KUKA KRL program: EPS_2_251529_SANMH_A_20250926032654.src

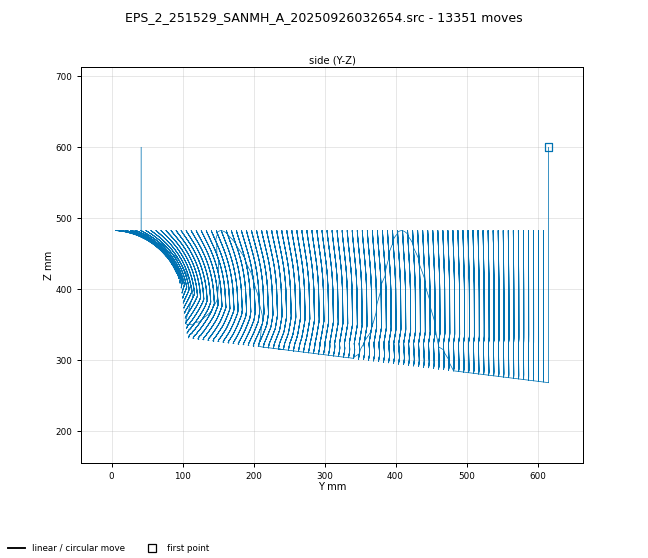
[picture p0: tool path of EPS_2_251529_SANMH_A_20250926032654.src, 13351 of 13353 moves have a stored position in this frame; points joined in program order, loops and branches not executed]
&ACCESS RVP
&REL 4
&COMMENT QRS 19112012
&PARAM EDITMASK = *
DEF PART()
EXT BAS (BAS_COMMAND :IN,REAL :IN )
INT I
BAS (#INITMOV,0 )

;KUKA QRS Post kuka4.cps  Date:22-06-2017 !

File_ID=2851

QRS_PRE_INIT()

;Init var - Until changes are made in qrs_pre_init
Outlet_Square_prg=0
Inlet_1_Square_prg=0
Inlet_2_Square_prg=0
Inlet_3_Square_prg=0
Inlet_4_Square_prg=0
Inlet_5_Square_prg=0

Outlet_1={X 0.000, Y 541.230, Z 408.000, B 0.000, E1 0.000 }
Inlet_1={X 0.000, Y 541.230, Z 408.000, B 0.000, E1 180.000 }
Outlet_1_type=150
Inlet_1_type=150
;QRS#1=Sidecore dimensions
;QRS#2=150-6" PVC SDR 28
;QRS#3=150-6" PVC SDR 28
;QRS#4=
;QRS#5=
;QRS#6=
;QRS#7=
;QRS#8=
;QRS#9=10-06 PSX
;QRS#10=10-06 PSX
;QRS#11=
;QRS#12=
;QRS#13=
;QRS#14=
;QRS#15=
;QRS#16=1220x127x762 2,5'
;QRS#17=EPS Height
;QRS#18=483
;QRS#19=*
;QRS#20= UPDATED VERSION 22-06-2017
;QRS#21=*
Outlet_Square=070
Inlet_1_Square=070
Inlet_2_Square=0
Inlet_3_Square=0
Inlet_4_Square=0
Inlet_5_Square=0
Mill_Square=1
Outlet_Square_Prg=203
Inlet_1_Square_prg=203

QRS_INIT()

$ADVANCE=5

; T1
PTP {E1 173.65,E2 173.65}
PTP {X 0,Y 615.436,A -85,B 0,C 180,E1 173.65,E2 173.65,E3 0,E4 0,E5 0,E6 0}
QRS_SPEED_INIT()
LIN {X 0,Y 615.436,Z 600,A -85,B 0,C 180,E1 173.65,E2 173.65,E3 0,E4 0,E5 0,E6 0} C_VEL
LIN {X 0,Y 615.436,Z 278.69,A -85,B 0,C 180,E1 173.65,E2 173.65} C_VEL
LIN {X 0,Y 615.436,Z 270.512,A -85,B 0,C 180,E1 173.65,E2 173.65} C_VEL
LIN {X 0,Y 615.421,Z 268.512,A -85,B 0,C 180,E1 173.464,E2 173.464} C_VEL
LIN {X 0,Y 615.418,Z 268.512,A -85,B 0,C 180,E1 171.462,E2 171.462} C_VEL
LIN {X 0,Y 615.412,Z 268.512,A -85,B 0,C 180,E1 169.141,E2 169.141} C_VEL
LIN {X 0,Y 615.434,Z 268.512,A -85,B 0,C 180,E1 166.798,E2 166.798} C_VEL
LIN {X 0,Y 615.46,Z 268.512,A -85,B 0,C 180,E1 164.094,E2 164.094} C_VEL
LIN {X 0,Y 615.413,Z 268.512,A -85,B 0,C 180,E1 161.352,E2 161.352} C_VEL
LIN {X 0,Y 615.489,Z 268.512,A -85,B 0,C 180,E1 158.568,E2 158.568} C_VEL
LIN {X 0,Y 615.416,Z 268.512,A -85,B 0,C 180,E1 155.725,E2 155.725} C_VEL
LIN {X 0,Y 615.415,Z 268.512,A -85,B 0,C 180,E1 153.552,E2 153.552} C_VEL
LIN {X 0,Y 615.478,Z 268.514,A -85,B 0,C 180,E1 150.593,E2 150.593} C_VEL
LIN {X 0,Y 615.446,Z 268.511,A -85,B 0,C 180,E1 148.312,E2 148.312} C_VEL
LIN {X 0,Y 615.418,Z 268.511,A -85,B 0,C 180,E1 145.974,E2 145.974} C_VEL
LIN {X 0,Y 615.472,Z 268.512,A -85,B 0,C 180,E1 143.064,E2 143.064} C_VEL
LIN {X 0,Y 615.424,Z 268.511,A -85,B 0,C 180,E1 140.245,E2 140.245} C_VEL
LIN {X 0,Y 615.417,Z 268.511,A -85,B 0,C 180,E1 137.926,E2 137.926} C_VEL
LIN {X 0,Y 615.42,Z 268.512,A -85,B 0,C 180,E1 135.844,E2 135.844} C_VEL
LIN {X 0,Y 615.48,Z 268.512,A -85,B 0,C 180,E1 133.244,E2 133.244} C_VEL
LIN {X 0,Y 615.438,Z 268.51,A -85,B 0,C 180,E1 130.609,E2 130.609} C_VEL
LIN {X 0,Y 615.466,Z 268.51,A -85,B 0,C 180,E1 128.905,E2 128.905} C_VEL
LIN {X 0,Y 615.423,Z 268.51,A -85,B 0,C 180,E1 126.428,E2 126.428} C_VEL
LIN {X 0,Y 615.471,Z 268.513,A -85,B 0,C 180,E1 123.532,E2 123.532} C_VEL
LIN {X 0,Y 615.448,Z 268.509,A -85,B 0,C 180,E1 120.921,E2 120.921} C_VEL
LIN {X 0,Y 615.421,Z 268.51,A -85,B 0,C 180,E1 118.439,E2 118.439} C_VEL
LIN {X 0,Y 615.474,Z 268.512,A -85,B 0,C 180,E1 115.716,E2 115.716} C_VEL
LIN {X 0,Y 615.43,Z 268.509,A -85,B 0,C 180,E1 112.846,E2 112.846} C_VEL
LIN {X 0,Y 615.423,Z 268.51,A -85,B 0,C 180,E1 110.54,E2 110.54} C_VEL
LIN {X 0,Y 615.492,Z 268.765,A -85,B 0,C 180,E1 109.598,E2 109.598} C_VEL
LIN {X 0,Y 615.471,Z 283.781,A -85,B 0,C 180,E1 106.928,E2 106.928} C_VEL
LIN {X 0,Y 615.47,Z 299.164,A -85,B 0,C 180,E1 104.241,E2 104.241} C_VEL
LIN {X 0,Y 615.494,Z 314.868,A -85,B 0,C 180,E1 101.526,E2 101.526} C_VEL
LIN {X 0,Y 615.495,Z 323.333,A -85,B 0,C 180,E1 100.111,E2 100.111} C_VEL
LIN {X 0,Y 615.495,Z 324.837,A -85,B 0,C 180,E1 100.049,E2 100.049} C_VEL
LIN {X 0,Y 615.492,Z 399.723,A -85,B 0,C 180,E1 99.157,E2 99.157} C_VEL
LIN {X 0,Y 615.496,Z 407.902,A -85,B 0,C 180,E1 98.991,E2 98.991} C_VEL
LIN {X 0,Y 615.497,Z 416.457,A -85,B 0,C 180,E1 98.743,E2 98.743} C_VEL
LIN {X 0,Y 615.497,Z 424.066,A -85,B 0,C 180,E1 98.454,E2 98.454} C_VEL
LIN {X 0,Y 615.499,Z 432.585,A -85,B 0,C 180,E1 98.04,E2 98.04} C_VEL
LIN {X 0,Y 615.487,Z 440.752,A -85,B 0,C 180,E1 97.545,E2 97.545} C_VEL
LIN {X 0,Y 615.492,Z 447.39,A -85,B 0,C 180,E1 97.058,E2 97.058} C_VEL
LIN {X 0,Y 615.498,Z 453.186,A -85,B 0,C 180,E1 96.556,E2 96.556} C_VEL
LIN {X 0,Y 615.499,Z 459.536,A -85,B 0,C 180,E1 95.898,E2 95.898} C_VEL
LIN {X 0,Y 615.495,Z 465.985,A -85,B 0,C 180,E1 95.077,E2 95.077} C_VEL
LIN {X 0,Y 615.491,Z 471.123,A -85,B 0,C 180,E1 94.256,E2 94.256} C_VEL
LIN {X 0,Y 615.493,Z 475.887,A -85,B 0,C 180,E1 93.273,E2 93.273} C_VEL
LIN {X 0,Y 615.493,Z 478.2,A -85,B 0,C 180,E1 92.618,E2 92.618} C_VEL
LIN {X 0,Y 615.5,Z 479.976,A -85,B 0,C 180,E1 91.963,E2 91.963} C_VEL
LIN {X 0,Y 615.492,Z 481.266,A -85,B 0,C 180,E1 91.309,E2 91.309} C_VEL
LIN {X 0,Y 615.491,Z 482.084,A -85,B 0,C 180,E1 90.654,E2 90.654} C_VEL
LIN {X 0,Y 615.492,Z 482.384,A -85,B 0,C 180,E1 90,E2 90} C_VEL
LIN {X 0,Y 615.492,Z 482.125,A -85,B 0,C 180,E1 89.346,E2 89.346} C_VEL
LIN {X 0,Y 615.494,Z 481.394,A -85,B 0,C 180,E1 88.691,E2 88.691} C_VEL
LIN {X 0,Y 615.5,Z 480.194,A -85,B 0,C 180,E1 88.037,E2 88.037} C_VEL
LIN {X 0,Y 615.49,Z 477.376,A -85,B 0,C 180,E1 87.055,E2 87.055} C_VEL
LIN {X 0,Y 615.492,Z 474.81,A -85,B 0,C 180,E1 86.399,E2 86.399} C_VEL
LIN {X 0,Y 615.495,Z 469.743,A -85,B 0,C 180,E1 85.416,E2 85.416} C_VEL
LIN {X 0,Y 615.496,Z 464.288,A -85,B 0,C 180,E1 84.595,E2 84.595} C_VEL
LIN {X 0,Y 615.497,Z 457.454,A -85,B 0,C 180,E1 83.773,E2 83.773} C_VEL
LIN {X 0,Y 615.497,Z 450.42,A -85,B 0,C 180,E1 83.1,E2 83.1} C_VEL
LIN {X 0,Y 615.487,Z 442.074,A -85,B 0,C 180,E1 82.455,E2 82.455} C_VEL
LIN {X 0,Y 615.499,Z 434.197,A -85,B 0,C 180,E1 81.96,E2 81.96} C_VEL
LIN {X 0,Y 615.497,Z 426.076,A -85,B 0,C 180,E1 81.546,E2 81.546} C_VEL
LIN {X 0,Y 615.497,Z 417.865,A -85,B 0,C 180,E1 81.216,E2 81.216} C_VEL
LIN {X 0,Y 615.497,Z 409.844,A -85,B 0,C 180,E1 80.967,E2 80.967} C_VEL
LIN {X 0,Y 615.497,Z 400.169,A -85,B 0,C 180,E1 80.76,E2 80.76} C_VEL
LIN {X 0,Y 615.493,Z 324.19,A -85,B 0,C 180,E1 79.848,E2 79.848} C_VEL
LIN {X 0,Y 615.49,Z 322.717,A -85,B 0,C 180,E1 79.723,E2 79.723} C_VEL
LIN {X 0,Y 615.485,Z 307.623,A -85,B 0,C 180,E1 77.135,E2 77.135} C_VEL
LIN {X 0,Y 615.491,Z 292.071,A -85,B 0,C 180,E1 74.435,E2 74.435} C_VEL
LIN {X 0,Y 615.479,Z 276.618,A -85,B 0,C 180,E1 71.719,E2 71.719} C_VEL
LIN {X 0,Y 615.493,Z 268.624,A -85,B 0,C 180,E1 70.272,E2 70.272} C_VEL
LIN {X 0,Y 615.436,Z 268.51,A -85,B 0,C 180,E1 67.666,E2 67.666} C_VEL
LIN {X 0,Y 615.437,Z 268.51,A -85,B 0,C 180,E1 65.726,E2 65.726} C_VEL
LIN {X 0,Y 615.427,Z 268.509,A -85,B 0,C 180,E1 63.554,E2 63.554} C_VEL
LIN {X 0,Y 615.431,Z 268.508,A -85,B 0,C 180,E1 61.34,E2 61.34} C_VEL
LIN {X 0,Y 615.469,Z 268.507,A -85,B 0,C 180,E1 58.917,E2 58.917} C_VEL
LIN {X 0,Y 615.435,Z 268.51,A -85,B 0,C 180,E1 55.976,E2 55.976} C_VEL
LIN {X 0,Y 615.428,Z 268.509,A -85,B 0,C 180,E1 53.572,E2 53.572} C_VEL
LIN {X 0,Y 615.49,Z 268.507,A -85,B 0,C 180,E1 50.938,E2 50.938} C_VEL
LIN {X 0,Y 615.467,Z 268.512,A -85,B 0,C 180,E1 48.526,E2 48.526} C_VEL
LIN {X 0,Y 615.425,Z 268.51,A -85,B 0,C 180,E1 46.009,E2 46.009} C_VEL
LIN {X 0,Y 615.424,Z 268.51,A -85,B 0,C 180,E1 43.993,E2 43.993} C_VEL
LIN {X 0,Y 615.449,Z 268.508,A -85,B 0,C 180,E1 41.477,E2 41.477} C_VEL
LIN {X 0,Y 615.485,Z 268.512,A -85,B 0,C 180,E1 38.905,E2 38.905} C_VEL
LIN {X 0,Y 615.43,Z 268.511,A -85,B 0,C 180,E1 36.429,E2 36.429} C_VEL
LIN {X 0,Y 615.422,Z 268.51,A -85,B 0,C 180,E1 34.026,E2 34.026} C_VEL
LIN {X 0,Y 615.445,Z 268.51,A -85,B 0,C 180,E1 31.688,E2 31.688} C_VEL
LIN {X 0,Y 615.479,Z 268.511,A -85,B 0,C 180,E1 29.407,E2 29.407} C_VEL
LIN {X 0,Y 615.42,Z 268.511,A -85,B 0,C 180,E1 26.447,E2 26.447} C_VEL
LIN {X 0,Y 615.435,Z 268.51,A -85,B 0,C 180,E1 24,E2 24} C_VEL
LIN {X 0,Y 615.498,Z 268.513,A -85,B 0,C 180,E1 21.432,E2 21.432} C_VEL
LIN {X 0,Y 615.415,Z 268.512,A -85,B 0,C 180,E1 18.589,E2 18.589} C_VEL
LIN {X 0,Y 615.462,Z 268.51,A -85,B 0,C 180,E1 15.906,E2 15.906} C_VEL
LIN {X 0,Y 615.441,Z 268.512,A -85,B 0,C 180,E1 13.202,E2 13.202} C_VEL
LIN {X 0,Y 615.417,Z 268.512,A -85,B 0,C 180,E1 10.861,E2 10.861} C_VEL
LIN {X 0,Y 615.421,Z 268.511,A -85,B 0,C 180,E1 8.538,E2 8.538} C_VEL
LIN {X 0,Y 615.496,Z 268.511,A -85,B 0,C 180,E1 5.899,E2 5.899} C_VEL
LIN {X 0,Y 615.426,Z 268.512,A -85,B 0,C 180,E1 3.273,E2 3.273} C_VEL
LIN {X 0,Y 615.425,Z 268.512,A -85,B 0,C 180,E1 1.309,E2 1.309} C_VEL
LIN {X 0,Y 615.423,Z 268.512,A -85,B 0,C 180,E1 -0.654,E2 -0.654} C_VEL
LIN {X 0,Y 615.42,Z 268.513,A -85,B 0,C 180,E1 -2.618,E2 -2.618} C_VEL
LIN {X 0,Y 615.42,Z 268.513,A -85,B 0,C 180,E1 -4.585,E2 -4.585} C_VEL
LIN {X 0,Y 615.42,Z 268.512,A -85,B 0,C 180,E1 -6.557,E2 -6.557} C_VEL
LIN {X 0,Y 615.418,Z 268.512,A -85,B 0,C 180,E1 -8.538,E2 -8.538} C_VEL
LIN {X 0,Y 615.413,Z 268.512,A -85,B 0,C 180,E1 -10.859,E2 -10.859} C_VEL
LIN {X 0,Y 615.435,Z 268.512,A -85,B 0,C 180,E1 -13.202,E2 -13.202} C_VEL
LIN {X 0,Y 615.46,Z 268.512,A -85,B 0,C 180,E1 -15.906,E2 -15.906} C_VEL
LIN {X 0,Y 615.414,Z 268.512,A -85,B 0,C 180,E1 -18.648,E2 -18.648} C_VEL
LIN {X 0,Y 615.491,Z 268.512,A -85,B 0,C 180,E1 -21.432,E2 -21.432} C_VEL
LIN {X 0,Y 615.418,Z 268.512,A -85,B 0,C 180,E1 -24.275,E2 -24.275} C_VEL
LIN {X 0,Y 615.416,Z 268.512,A -85,B 0,C 180,E1 -26.447,E2 -26.447} C_VEL
LIN {X 0,Y 615.479,Z 268.513,A -85,B 0,C 180,E1 -29.407,E2 -29.407} C_VEL
LIN {X 0,Y 615.447,Z 268.51,A -85,B 0,C 180,E1 -31.688,E2 -31.688} C_VEL
LIN {X 0,Y 615.421,Z 268.511,A -85,B 0,C 180,E1 -34.026,E2 -34.026} C_VEL
LIN {X 0,Y 615.475,Z 268.512,A -85,B 0,C 180,E1 -36.937,E2 -36.937} C_VEL
LIN {X 0,Y 615.426,Z 268.511,A -85,B 0,C 180,E1 -39.755,E2 -39.755} C_VEL
LIN {X 0,Y 615.42,Z 268.511,A -85,B 0,C 180,E1 -42.075,E2 -42.075} C_VEL
LIN {X 0,Y 615.423,Z 268.511,A -85,B 0,C 180,E1 -44.155,E2 -44.155} C_VEL
LIN {X 0,Y 615.485,Z 268.512,A -85,B 0,C 180,E1 -46.756,E2 -46.756} C_VEL
LIN {X 0,Y 615.44,Z 268.509,A -85,B 0,C 180,E1 -49.391,E2 -49.391} C_VEL
LIN {X 0,Y 615.467,Z 268.509,A -85,B 0,C 180,E1 -51.095,E2 -51.095} C_VEL
LIN {X 0,Y 615.425,Z 268.51,A -85,B 0,C 180,E1 -53.572,E2 -53.572} C_VEL
LIN {X 0,Y 615.479,Z 268.512,A -85,B 0,C 180,E1 -56.467,E2 -56.467} C_VEL
LIN {X 0,Y 615.449,Z 268.508,A -85,B 0,C 180,E1 -59.079,E2 -59.079} C_VEL
LIN {X 0,Y 615.424,Z 268.51,A -85,B 0,C 180,E1 -61.561,E2 -61.561} C_VEL
LIN {X 0,Y 615.498,Z 268.512,A -85,B 0,C 180,E1 -64.429,E2 -64.429} C_VEL
LIN {X 0,Y 615.432,Z 268.509,A -85,B 0,C 180,E1 -67.154,E2 -67.154} C_VEL
LIN {X 0,Y 615.427,Z 268.51,A -85,B 0,C 180,E1 -69.458,E2 -69.458} C_VEL
LIN {X 0,Y 615.492,Z 268.773,A -85,B 0,C 180,E1 -70.359,E2 -70.359} C_VEL
LIN {X 0,Y 615.469,Z 284.037,A -85,B 0,C 180,E1 -73.072,E2 -73.072} C_VEL
LIN {X 0,Y 615.471,Z 299.417,A -85,B 0,C 180,E1 -75.758,E2 -75.758} C_VEL
LIN {X 0,Y 615.492,Z 315.131,A -85,B 0,C 180,E1 -78.474,E2 -78.474} C_VEL
LIN {X 0,Y 615.494,Z 323.371,A -85,B 0,C 180,E1 -79.848,E2 -79.848} C_VEL
LIN {X 0,Y 615.494,Z 325.037,A -85,B 0,C 180,E1 -79.91,E2 -79.91} C_VEL
LIN {X 0,Y 615.494,Z 399.946,A -85,B 0,C 180,E1 -80.802,E2 -80.802} C_VEL
LIN {X 0,Y 615.497,Z 409.7,A -85,B 0,C 180,E1 -81.009,E2 -81.009} C_VEL
LIN {X 0,Y 615.499,Z 420.157,A -85,B 0,C 180,E1 -81.34,E2 -81.34} C_VEL
LIN {X 0,Y 615.497,Z 430.43,A -85,B 0,C 180,E1 -81.794,E2 -81.794} C_VEL
LIN {X 0,Y 615.489,Z 440.201,A -85,B 0,C 180,E1 -82.372,E2 -82.372} C_VEL
LIN {X 0,Y 615.494,Z 447.936,A -85,B 0,C 180,E1 -82.942,E2 -82.942} C_VEL
LIN {X 0,Y 615.497,Z 455.335,A -85,B 0,C 180,E1 -83.608,E2 -83.608} C_VEL
LIN {X 0,Y 615.498,Z 462.738,A -85,B 0,C 180,E1 -84.43,E2 -84.43} C_VEL
LIN {X 0,Y 615.497,Z 468.533,A -85,B 0,C 180,E1 -85.252,E2 -85.252} C_VEL
LIN {X 0,Y 615.496,Z 473.1,A -85,B 0,C 180,E1 -86.072,E2 -86.072} C_VEL
LIN {X 0,Y 615.492,Z 476.069,A -85,B 0,C 180,E1 -86.727,E2 -86.727} C_VEL
LIN {X 0,Y 615.494,Z 478.357,A -85,B 0,C 180,E1 -87.382,E2 -87.382} C_VEL
LIN {X 0,Y 615.5,Z 480.085,A -85,B 0,C 180,E1 -88.037,E2 -88.037} C_VEL
LIN {X 0,Y 615.493,Z 481.33,A -85,B 0,C 180,E1 -88.691,E2 -88.691} C_VEL
LIN {X 0,Y 615.491,Z 482.104,A -85,B 0,C 180,E1 -89.346,E2 -89.346} C_VEL
LIN {X 0,Y 615.491,Z 482.389,A -85,B 0,C 180,E1 -90,E2 -90} C_VEL
LIN {X 0,Y 615.491,Z 482.104,A -85,B 0,C 180,E1 -90.654,E2 -90.654} C_VEL
LIN {X 0,Y 615.493,Z 481.33,A -85,B 0,C 180,E1 -91.309,E2 -91.309} C_VEL
LIN {X 0,Y 615.5,Z 480.085,A -85,B 0,C 180,E1 -91.963,E2 -91.963} C_VEL
LIN {X 0,Y 615.488,Z 477.221,A -85,B 0,C 180,E1 -92.945,E2 -92.945} C_VEL
LIN {X 0,Y 615.491,Z 474.604,A -85,B 0,C 180,E1 -93.601,E2 -93.601} C_VEL
LIN {X 0,Y 615.495,Z 469.483,A -85,B 0,C 180,E1 -94.584,E2 -94.584} C_VEL
LIN {X 0,Y 615.495,Z 463.969,A -85,B 0,C 180,E1 -95.405,E2 -95.405} C_VEL
LIN {X 0,Y 615.498,Z 457.019,A -85,B 0,C 180,E1 -96.227,E2 -96.227} C_VEL
LIN {X 0,Y 615.496,Z 449.86,A -85,B 0,C 180,E1 -96.901,E2 -96.901} C_VEL
LIN {X 0,Y 615.485,Z 442.625,A -85,B 0,C 180,E1 -97.463,E2 -97.463} C_VEL
LIN {X 0,Y 615.497,Z 434.871,A -85,B 0,C 180,E1 -97.958,E2 -97.958} C_VEL
LIN {X 0,Y 615.498,Z 426.917,A -85,B 0,C 180,E1 -98.371,E2 -98.371} C_VEL
LIN {X 0,Y 615.497,Z 417.76,A -85,B 0,C 180,E1 -98.743,E2 -98.743} C_VEL
LIN {X 0,Y 615.497,Z 409.7,A -85,B 0,C 180,E1 -98.991,E2 -98.991} C_VEL
LIN {X 0,Y 615.494,Z 399.946,A -85,B 0,C 180,E1 -99.198,E2 -99.198} C_VEL
LIN {X 0,Y 615.494,Z 324.09,A -85,B 0,C 180,E1 -100.111,E2 -100.111} C_VEL
LIN {X 0,Y 615.492,Z 322.973,A -85,B 0,C 180,E1 -100.194,E2 -100.194} C_VEL
LIN {X 0,Y 615.48,Z 307.363,A -85,B 0,C 180,E1 -102.865,E2 -102.865} C_VEL
LIN {X 0,Y 615.49,Z 291.813,A -85,B 0,C 180,E1 -105.565,E2 -105.565} C_VEL
LIN {X 0,Y 615.482,Z 276.36,A -85,B 0,C 180,E1 -108.282,E2 -108.282} C_VEL
LIN {X 0,Y 615.49,Z 268.621,A -85,B 0,C 180,E1 -109.684,E2 -109.684} C_VEL
LIN {X 0,Y 615.432,Z 268.51,A -85,B 0,C 180,E1 -112.333,E2 -112.333} C_VEL
LIN {X 0,Y 615.432,Z 268.51,A -85,B 0,C 180,E1 -114.274,E2 -114.274} C_VEL
LIN {X 0,Y 615.424,Z 268.51,A -85,B 0,C 180,E1 -116.446,E2 -116.446} C_VEL
LIN {X 0,Y 615.492,Z 268.511,A -85,B 0,C 180,E1 -119.405,E2 -119.405} C_VEL
LIN {X 0,Y 615.466,Z 268.512,A -85,B 0,C 180,E1 -121.686,E2 -121.686} C_VEL
LIN {X 0,Y 615.431,Z 268.511,A -85,B 0,C 180,E1 -124.025,E2 -124.025} C_VEL
LIN {X 0,Y 615.426,Z 268.509,A -85,B 0,C 180,E1 -126.428,E2 -126.428} C_VEL
LIN {X 0,Y 615.49,Z 268.508,A -85,B 0,C 180,E1 -129.062,E2 -129.062} C_VEL
LIN {X 0,Y 615.462,Z 268.512,A -85,B 0,C 180,E1 -131.475,E2 -131.475} C_VEL
LIN {X 0,Y 615.423,Z 268.51,A -85,B 0,C 180,E1 -133.991,E2 -133.991} C_VEL
LIN {X 0,Y 615.422,Z 268.51,A -85,B 0,C 180,E1 -136.008,E2 -136.008} C_VEL
LIN {X 0,Y 615.447,Z 268.509,A -85,B 0,C 180,E1 -138.523,E2 -138.523} C_VEL
LIN {X 0,Y 615.481,Z 268.512,A -85,B 0,C 180,E1 -141.095,E2 -141.095} C_VEL
LIN {X 0,Y 615.428,Z 268.511,A -85,B 0,C 180,E1 -143.571,E2 -143.571} C_VEL
LIN {X 0,Y 615.422,Z 268.51,A -85,B 0,C 180,E1 -145.974,E2 -145.974} C_VEL
LIN {X 0,Y 615.444,Z 268.51,A -85,B 0,C 180,E1 -148.312,E2 -148.312} C_VEL
LIN {X 0,Y 615.478,Z 268.512,A -85,B 0,C 180,E1 -150.593,E2 -150.593} C_VEL
LIN {X 0,Y 615.419,Z 268.511,A -85,B 0,C 180,E1 -153.553,E2 -153.553} C_VEL
LIN {X 0,Y 615.433,Z 268.511,A -85,B 0,C 180,E1 -156,E2 -156} C_VEL
LIN {X 0,Y 615.497,Z 268.512,A -85,B 0,C 180,E1 -158.569,E2 -158.569} C_VEL
LIN {X 0,Y 615.415,Z 268.512,A -85,B 0,C 180,E1 -161.411,E2 -161.411} C_VEL
LIN {X 0,Y 615.462,Z 268.511,A -85,B 0,C 180,E1 -164.094,E2 -164.094} C_VEL
LIN {X 0,Y 615.44,Z 268.512,A -85,B 0,C 180,E1 -166.798,E2 -166.798} C_VEL
LIN {X 0,Y 615.417,Z 268.512,A -85,B 0,C 180,E1 -169.139,E2 -169.139} C_VEL
LIN {X 0,Y 615.421,Z 268.512,A -85,B 0,C 180,E1 -171.463,E2 -171.463} C_VEL
LIN {X 0,Y 615.496,Z 268.511,A -85,B 0,C 180,E1 -174.102,E2 -174.102} C_VEL
LIN {X 0,Y 615.426,Z 268.512,A -85,B 0,C 180,E1 -176.727,E2 -176.727} C_VEL
LIN {X 0,Y 615.425,Z 268.512,A -85,B 0,C 180,E1 -178.691,E2 -178.691} C_VEL
LIN {X 0,Y 615.423,Z 268.512,A -85,B 0,C 180,E1 -180.654,E2 -180.654} C_VEL
LIN {X 0,Y 615.42,Z 268.513,A -85,B 0,C 180,E1 -182.618,E2 -182.618} C_VEL
LIN {X 0,Y 615.421,Z 268.512,A -85,B 0,C 180,E1 -184.585,E2 -184.585} C_VEL
LIN {X 0,Y 615.421,Z 268.512,A -85,B 0,C 180,E1 -186.536,E2 -186.536} C_VEL
LIN {X 0,Y 614.744,Z 268.659,A -85,B 0,C 180,E1 -187.082,E2 -187.082} C_VEL
LIN {X 0,Y 611.908,Z 269.078,A -85,B 0,C 180,E1 -187.968,E2 -187.968} C_VEL
LIN {X 0,Y 609.524,Z 269.383,A -85,B 0,C 180,E1 -188.681,E2 -188.681} C_VEL
LIN {X 0,Y 608.503,Z 269.498,A -85,B 0,C 180,E1 -189.231,E2 -189.231} C_VEL
LIN {X 0,Y 608.421,Z 269.507,A -85,B 0,C 180,E1 -189.417,E2 -189.417} C_VEL
LIN {X 0,Y 608.436,Z 269.508,A -85,B 0,C 180,E1 -192,E2 -192} C_VEL
LIN {X 0,Y 608.385,Z 269.508,A -85,B 0,C 180,E1 -194.723,E2 -194.723} C_VEL
LIN {X 0,Y 608.418,Z 269.513,A -85,B 0,C 180,E1 -197.478,E2 -197.478} C_VEL
LIN {X 0,Y 608.405,Z 269.507,A -85,B 0,C 180,E1 -200.276,E2 -200.276} C_VEL
LIN {X 0,Y 608.385,Z 269.508,A -85,B 0,C 180,E1 -202.463,E2 -202.463} C_VEL
LIN {X 0,Y 608.403,Z 269.506,A -85,B 0,C 180,E1 -204.573,E2 -204.573} C_VEL
LIN {X 0,Y 608.458,Z 269.507,A -85,B 0,C 180,E1 -207.206,E2 -207.206} C_VEL
LIN {X 0,Y 608.401,Z 269.508,A -85,B 0,C 180,E1 -209.963,E2 -209.963} C_VEL
LIN {X 0,Y 608.404,Z 269.507,A -85,B 0,C 180,E1 -212.516,E2 -212.516} C_VEL
LIN {X 0,Y 608.414,Z 269.511,A -85,B 0,C 180,E1 -214.903,E2 -214.903} C_VEL
LIN {X 0,Y 608.425,Z 269.505,A -85,B 0,C 180,E1 -217.75,E2 -217.75} C_VEL
LIN {X 0,Y 608.393,Z 269.508,A -85,B 0,C 180,E1 -220.324,E2 -220.324} C_VEL
LIN {X 0,Y 608.443,Z 269.512,A -85,B 0,C 180,E1 -222.961,E2 -222.961} C_VEL
LIN {X 0,Y 608.401,Z 269.507,A -85,B 0,C 180,E1 -225.742,E2 -225.742} C_VEL
LIN {X 0,Y 608.403,Z 269.506,A -85,B 0,C 180,E1 -227.935,E2 -227.935} C_VEL
LIN {X 0,Y 608.432,Z 269.512,A -85,B 0,C 180,E1 -230.707,E2 -230.707} C_VEL
LIN {X 0,Y 608.433,Z 269.507,A -85,B 0,C 180,E1 -233.084,E2 -233.084} C_VEL
LIN {X 0,Y 608.42,Z 269.504,A -85,B 0,C 180,E1 -235.528,E2 -235.528} C_VEL
LIN {X 0,Y 608.418,Z 269.505,A -85,B 0,C 180,E1 -237.904,E2 -237.904} C_VEL
LIN {X 0,Y 608.438,Z 269.507,A -85,B 0,C 180,E1 -240.22,E2 -240.22} C_VEL
LIN {X 0,Y 608.399,Z 269.507,A -85,B 0,C 180,E1 -243.224,E2 -243.224} C_VEL
LIN {X 0,Y 608.409,Z 269.505,A -85,B 0,C 180,E1 -245.428,E2 -245.428} C_VEL
LIN {X 0,Y 608.452,Z 269.51,A -85,B 0,C 180,E1 -248.308,E2 -248.308} C_VEL
LIN {X 0,Y 608.478,Z 269.608,A -85,B 0,C 180,E1 -250.299,E2 -250.299} C_VEL
LIN {X 0,Y 608.508,Z 281.933,A -85,B 0,C 180,E1 -252.526,E2 -252.526} C_VEL
LIN {X 0,Y 608.472,Z 297.545,A -85,B 0,C 180,E1 -255.28,E2 -255.28} C_VEL
LIN {X 0,Y 608.463,Z 313.158,A -85,B 0,C 180,E1 -258.001,E2 -258.001} C_VEL
LIN {X 0,Y 608.483,Z 323.536,A -85,B 0,C 180,E1 -259.771,E2 -259.771} C_VEL
LIN {X 0,Y 608.517,Z 325.183,A -85,B 0,C 180,E1 -259.835,E2 -259.835} C_VEL
LIN {X 0,Y 608.507,Z 400.265,A -85,B 0,C 180,E1 -260.737,E2 -260.737} C_VEL
LIN {X 0,Y 608.51,Z 409.96,A -85,B 0,C 180,E1 -260.946,E2 -260.946} C_VEL
LIN {X 0,Y 608.499,Z 421.543,A -85,B 0,C 180,E1 -261.323,E2 -261.323} C_VEL
LIN {X 0,Y 608.479,Z 431.436,A -85,B 0,C 180,E1 -261.783,E2 -261.783} C_VEL
LIN {X 0,Y 608.47,Z 439.888,A -85,B 0,C 180,E1 -262.284,E2 -262.284} C_VEL
LIN {X 0,Y 608.46,Z 447.856,A -85,B 0,C 180,E1 -262.867,E2 -262.867} C_VEL
LIN {X 0,Y 608.467,Z 454.903,A -85,B 0,C 180,E1 -263.496,E2 -263.496} C_VEL
LIN {X 0,Y 608.458,Z 461.397,A -85,B 0,C 180,E1 -264.2,E2 -264.2} C_VEL
LIN {X 0,Y 608.437,Z 467.642,A -85,B 0,C 180,E1 -265.03,E2 -265.03} C_VEL
LIN {X 0,Y 608.434,Z 473.425,A -85,B 0,C 180,E1 -266.026,E2 -266.026} C_VEL
LIN {X 0,Y 608.447,Z 477.631,A -85,B 0,C 180,E1 -267.021,E2 -267.021} C_VEL
LIN {X 0,Y 608.444,Z 480.57,A -85,B 0,C 180,E1 -268.014,E2 -268.014} C_VEL
LIN {X 0,Y 608.445,Z 481.87,A -85,B 0,C 180,E1 -268.676,E2 -268.676} C_VEL
LIN {X 0,Y 608.434,Z 482.692,A -85,B 0,C 180,E1 -269.338,E2 -269.338} C_VEL
LIN {X 0,Y 608.432,Z 482.995,A -85,B 0,C 180,E1 -270,E2 -270} C_VEL
LIN {X 0,Y 608.435,Z 482.735,A -85,B 0,C 180,E1 -270.662,E2 -270.662} C_VEL
LIN {X 0,Y 608.446,Z 481.997,A -85,B 0,C 180,E1 -271.324,E2 -271.324} C_VEL
LIN {X 0,Y 608.444,Z 480.787,A -85,B 0,C 180,E1 -271.986,E2 -271.986} C_VEL
LIN {X 0,Y 608.445,Z 477.942,A -85,B 0,C 180,E1 -272.979,E2 -272.979} C_VEL
LIN {X 0,Y 608.446,Z 475.352,A -85,B 0,C 180,E1 -273.642,E2 -273.642} C_VEL
LIN {X 0,Y 608.445,Z 470.245,A -85,B 0,C 180,E1 -274.638,E2 -274.638} C_VEL
LIN {X 0,Y 608.461,Z 464.749,A -85,B 0,C 180,E1 -275.468,E2 -275.468} C_VEL
LIN {X 0,Y 608.454,Z 457.149,A -85,B 0,C 180,E1 -276.374,E2 -276.374} C_VEL
LIN {X 0,Y 608.463,Z 448.95,A -85,B 0,C 180,E1 -277.132,E2 -277.132} C_VEL
LIN {X 0,Y 608.469,Z 441.201,A -85,B 0,C 180,E1 -277.716,E2 -277.716} C_VEL
LIN {X 0,Y 608.48,Z 433.036,A -85,B 0,C 180,E1 -278.217,E2 -278.217} C_VEL
LIN {X 0,Y 608.485,Z 422.678,A -85,B 0,C 180,E1 -278.719,E2 -278.719} C_VEL
LIN {X 0,Y 608.509,Z 411.036,A -85,B 0,C 180,E1 -279.116,E2 -279.116} C_VEL
LIN {X 0,Y 608.519,Z 400.649,A -85,B 0,C 180,E1 -279.347,E2 -279.347} C_VEL
LIN {X 0,Y 608.517,Z 361.351,A -85,B 0,C 180,E1 -279.829,E2 -279.829} C_VEL
LIN {X 0,Y 608.513,Z 324.373,A -85,B 0,C 180,E1 -280.27,E2 -280.27} C_VEL
LIN {X 0,Y 608.456,Z 323.249,A -85,B 0,C 180,E1 -280.355,E2 -280.355} C_VEL
LIN {X 0,Y 608.449,Z 307.821,A -85,B 0,C 180,E1 -283.017,E2 -283.017} C_VEL
LIN {X 0,Y 608.466,Z 292.202,A -85,B 0,C 180,E1 -285.749,E2 -285.749} C_VEL
LIN {X 0,Y 608.517,Z 275.404,A -85,B 0,C 180,E1 -288.728,E2 -288.728} C_VEL
LIN {X 0,Y 608.488,Z 269.568,A -85,B 0,C 180,E1 -289.811,E2 -289.811} C_VEL
LIN {X 0,Y 608.428,Z 269.503,A -85,B 0,C 180,E1 -292.469,E2 -292.469} C_VEL
LIN {X 0,Y 608.415,Z 269.505,A -85,B 0,C 180,E1 -294.572,E2 -294.572} C_VEL
LIN {X 0,Y 608.461,Z 269.503,A -85,B 0,C 180,E1 -297.204,E2 -297.204} C_VEL
LIN {X 0,Y 608.421,Z 269.507,A -85,B 0,C 180,E1 -299.964,E2 -299.964} C_VEL
LIN {X 0,Y 608.413,Z 269.505,A -85,B 0,C 180,E1 -302.515,E2 -302.515} C_VEL
LIN {X 0,Y 608.417,Z 269.507,A -85,B 0,C 180,E1 -304.901,E2 -304.901} C_VEL
LIN {X 0,Y 608.437,Z 269.506,A -85,B 0,C 180,E1 -307.748,E2 -307.748} C_VEL
LIN {X 0,Y 608.398,Z 269.507,A -85,B 0,C 180,E1 -310.323,E2 -310.323} C_VEL
LIN {X 0,Y 608.445,Z 269.507,A -85,B 0,C 180,E1 -312.959,E2 -312.959} C_VEL
LIN {X 0,Y 608.409,Z 269.507,A -85,B 0,C 180,E1 -315.739,E2 -315.739} C_VEL
LIN {X 0,Y 608.408,Z 269.506,A -85,B 0,C 180,E1 -317.934,E2 -317.934} C_VEL
LIN {X 0,Y 608.435,Z 269.508,A -85,B 0,C 180,E1 -320.705,E2 -320.705} C_VEL
LIN {X 0,Y 608.45,Z 269.509,A -85,B 0,C 180,E1 -323.085,E2 -323.085} C_VEL
LIN {X 0,Y 608.425,Z 269.505,A -85,B 0,C 180,E1 -325.528,E2 -325.528} C_VEL
LIN {X 0,Y 608.414,Z 269.505,A -85,B 0,C 180,E1 -327.902,E2 -327.902} C_VEL
LIN {X 0,Y 608.428,Z 269.505,A -85,B 0,C 180,E1 -330.218,E2 -330.218} C_VEL
LIN {X 0,Y 608.466,Z 269.507,A -85,B 0,C 180,E1 -332.792,E2 -332.792} C_VEL
LIN {X 0,Y 608.408,Z 269.506,A -85,B 0,C 180,E1 -335.427,E2 -335.427} C_VEL
LIN {X 0,Y 608.453,Z 269.506,A -85,B 0,C 180,E1 -338.308,E2 -338.308} C_VEL
LIN {X 0,Y 608.401,Z 269.507,A -85,B 0,C 180,E1 -341.299,E2 -341.299} C_VEL
LIN {X 0,Y 608.422,Z 269.506,A -85,B 0,C 180,E1 -343.905,E2 -343.905} C_VEL
LIN {X 0,Y 608.428,Z 269.509,A -85,B 0,C 180,E1 -346.643,E2 -346.643} C_VEL
LIN {X 0,Y 608.4,Z 269.507,A -85,B 0,C 180,E1 -349.349,E2 -349.349} C_VEL
LIN {X 0,Y 608.461,Z 269.506,A -85,B 0,C 180,E1 -352.033,E2 -352.033} C_VEL
LIN {X 0,Y 608.415,Z 269.507,A -85,B 0,C 180,E1 -354.698,E2 -354.698} C_VEL
LIN {X 0,Y 608.418,Z 269.505,A -85,B 0,C 180,E1 -357.352,E2 -357.352} C_VEL
LIN {X 0,Y 608.465,Z 269.509,A -85,B 0,C 180,E1 -360,E2 -360} C_VEL
LIN {X 0,Y 608.416,Z 269.506,A -85,B 0,C 180,E1 -362.648,E2 -362.648} C_VEL
LIN {X 0,Y 608.409,Z 269.507,A -85,B 0,C 180,E1 -365.302,E2 -365.302} C_VEL
LIN {X 0,Y 608.457,Z 269.507,A -85,B 0,C 180,E1 -367.967,E2 -367.967} C_VEL
LIN {X 0,Y 608.397,Z 269.507,A -85,B 0,C 180,E1 -370.651,E2 -370.651} C_VEL
LIN {X 0,Y 608.423,Z 269.509,A -85,B 0,C 180,E1 -373.357,E2 -373.357} C_VEL
LIN {X 0,Y 608.419,Z 269.507,A -85,B 0,C 180,E1 -376.095,E2 -376.095} C_VEL
LIN {X 0,Y 608.418,Z 269.505,A -85,B 0,C 180,E1 -378.871,E2 -378.871} C_VEL
LIN {X 0,Y 608.449,Z 269.507,A -85,B 0,C 180,E1 -381.692,E2 -381.692} C_VEL
LIN {X 0,Y 608.404,Z 269.506,A -85,B 0,C 180,E1 -384.573,E2 -384.573} C_VEL
LIN {X 0,Y 608.459,Z 269.507,A -85,B 0,C 180,E1 -387.206,E2 -387.206} C_VEL
LIN {X 0,Y 608.401,Z 269.508,A -85,B 0,C 180,E1 -389.963,E2 -389.963} C_VEL
LIN {X 0,Y 608.406,Z 269.507,A -85,B 0,C 180,E1 -392.516,E2 -392.516} C_VEL
LIN {X 0,Y 608.409,Z 269.514,A -85,B 0,C 180,E1 -395.28,E2 -395.28} C_VEL
LIN {X 0,Y 608.426,Z 269.504,A -85,B 0,C 180,E1 -397.749,E2 -397.749} C_VEL
LIN {X 0,Y 608.395,Z 269.508,A -85,B 0,C 180,E1 -400.324,E2 -400.324} C_VEL
LIN {X 0,Y 608.446,Z 269.512,A -85,B 0,C 180,E1 -402.96,E2 -402.96} C_VEL
LIN {X 0,Y 608.403,Z 269.506,A -85,B 0,C 180,E1 -405.741,E2 -405.741} C_VEL
LIN {X 0,Y 608.405,Z 269.506,A -85,B 0,C 180,E1 -407.935,E2 -407.935} C_VEL
LIN {X 0,Y 608.434,Z 269.512,A -85,B 0,C 180,E1 -410.707,E2 -410.707} C_VEL
LIN {X 0,Y 608.434,Z 269.506,A -85,B 0,C 180,E1 -413.085,E2 -413.085} C_VEL
LIN {X 0,Y 608.423,Z 269.504,A -85,B 0,C 180,E1 -415.529,E2 -415.529} C_VEL
LIN {X 0,Y 608.422,Z 269.505,A -85,B 0,C 180,E1 -417.904,E2 -417.904} C_VEL
LIN {X 0,Y 608.44,Z 269.507,A -85,B 0,C 180,E1 -420.22,E2 -420.22} C_VEL
LIN {X 0,Y 608.402,Z 269.507,A -85,B 0,C 180,E1 -423.224,E2 -423.224} C_VEL
LIN {X 0,Y 608.412,Z 269.505,A -85,B 0,C 180,E1 -425.428,E2 -425.428} C_VEL
LIN {X 0,Y 608.454,Z 269.51,A -85,B 0,C 180,E1 -428.308,E2 -428.308} C_VEL
LIN {X 0,Y 608.462,Z 269.612,A -85,B 0,C 180,E1 -430.255,E2 -430.255} C_VEL
LIN {X 0,Y 608.507,Z 282.186,A -85,B 0,C 180,E1 -432.525,E2 -432.525} C_VEL
LIN {X 0,Y 608.471,Z 297.802,A -85,B 0,C 180,E1 -435.28,E2 -435.28} C_VEL
LIN {X 0,Y 608.462,Z 313.418,A -85,B 0,C 180,E1 -438.001,E2 -438.001} C_VEL
LIN {X 0,Y 608.467,Z 323.568,A -85,B 0,C 180,E1 -439.729,E2 -439.729} C_VEL
LIN {X 0,Y 608.519,Z 325.353,A -85,B 0,C 180,E1 -439.793,E2 -439.793} C_VEL
LIN {X 0,Y 608.504,Z 399.158,A -85,B 0,C 180,E1 -440.674,E2 -440.674} C_VEL
LIN {X 0,Y 608.523,Z 408.422,A -85,B 0,C 180,E1 -440.863,E2 -440.863} C_VEL
LIN {X 0,Y 608.49,Z 416.893,A -85,B 0,C 180,E1 -441.114,E2 -441.114} C_VEL
LIN {X 0,Y 608.501,Z 425.393,A -85,B 0,C 180,E1 -441.448,E2 -441.448} C_VEL
LIN {X 0,Y 608.497,Z 433.722,A -85,B 0,C 180,E1 -441.866,E2 -441.866} C_VEL
LIN {X 0,Y 608.468,Z 441.762,A -85,B 0,C 180,E1 -442.367,E2 -442.367} C_VEL
LIN {X 0,Y 608.452,Z 449.416,A -85,B 0,C 180,E1 -442.951,E2 -442.951} C_VEL
LIN {X 0,Y 608.452,Z 457.439,A -85,B 0,C 180,E1 -443.7,E2 -443.7} C_VEL
LIN {X 0,Y 608.46,Z 464.431,A -85,B 0,C 180,E1 -444.532,E2 -444.532} C_VEL
LIN {X 0,Y 608.431,Z 469.985,A -85,B 0,C 180,E1 -445.362,E2 -445.362} C_VEL
LIN {X 0,Y 608.445,Z 475.146,A -85,B 0,C 180,E1 -446.358,E2 -446.358} C_VEL
LIN {X 0,Y 608.444,Z 477.786,A -85,B 0,C 180,E1 -447.021,E2 -447.021} C_VEL
LIN {X 0,Y 608.444,Z 480.678,A -85,B 0,C 180,E1 -448.014,E2 -448.014} C_VEL
LIN {X 0,Y 608.446,Z 481.934,A -85,B 0,C 180,E1 -448.676,E2 -448.676} C_VEL
LIN {X 0,Y 608.434,Z 482.714,A -85,B 0,C 180,E1 -449.338,E2 -449.338} C_VEL
LIN {X 0,Y 608.431,Z 483,A -85,B 0,C 180,E1 -450,E2 -450} C_VEL
LIN {X 0,Y 608.434,Z 482.714,A -85,B 0,C 180,E1 -450.662,E2 -450.662} C_VEL
LIN {X 0,Y 608.446,Z 481.934,A -85,B 0,C 180,E1 -451.324,E2 -451.324} C_VEL
LIN {X 0,Y 608.444,Z 480.678,A -85,B 0,C 180,E1 -451.986,E2 -451.986} C_VEL
LIN {X 0,Y 608.444,Z 477.786,A -85,B 0,C 180,E1 -452.979,E2 -452.979} C_VEL
LIN {X 0,Y 608.445,Z 475.146,A -85,B 0,C 180,E1 -453.642,E2 -453.642} C_VEL
LIN {X 0,Y 608.431,Z 469.985,A -85,B 0,C 180,E1 -454.638,E2 -454.638} C_VEL
LIN {X 0,Y 608.46,Z 464.43,A -85,B 0,C 180,E1 -455.468,E2 -455.468} C_VEL
LIN {X 0,Y 608.455,Z 456.67,A -85,B 0,C 180,E1 -456.376,E2 -456.376} C_VEL
LIN {X 0,Y 608.452,Z 449.417,A -85,B 0,C 180,E1 -457.049,E2 -457.049} C_VEL
LIN {X 0,Y 608.468,Z 441.762,A -85,B 0,C 180,E1 -457.633,E2 -457.633} C_VEL
LIN {X 0,Y 608.497,Z 433.722,A -85,B 0,C 180,E1 -458.134,E2 -458.134} C_VEL
LIN {X 0,Y 608.501,Z 425.393,A -85,B 0,C 180,E1 -458.552,E2 -458.552} C_VEL
LIN {X 0,Y 608.49,Z 416.894,A -85,B 0,C 180,E1 -458.886,E2 -458.886} C_VEL
LIN {X 0,Y 608.513,Z 407.593,A -85,B 0,C 180,E1 -459.158,E2 -459.158} C_VEL
LIN {X 0,Y 608.508,Z 396.56,A -85,B 0,C 180,E1 -459.368,E2 -459.368} C_VEL
LIN {X 0,Y 608.509,Z 324.273,A -85,B 0,C 180,E1 -460.228,E2 -460.228} C_VEL
LIN {X 0,Y 608.451,Z 323.229,A -85,B 0,C 180,E1 -460.313,E2 -460.313} C_VEL
LIN {X 0,Y 608.444,Z 307.562,A -85,B 0,C 180,E1 -463.017,E2 -463.017} C_VEL
LIN {X 0,Y 608.465,Z 291.946,A -85,B 0,C 180,E1 -465.749,E2 -465.749} C_VEL
LIN {X 0,Y 608.497,Z 276.715,A -85,B 0,C 180,E1 -468.45,E2 -468.45} C_VEL
LIN {X 0,Y 608.466,Z 269.569,A -85,B 0,C 180,E1 -469.767,E2 -469.767} C_VEL
LIN {X 0,Y 608.411,Z 269.504,A -85,B 0,C 180,E1 -472.465,E2 -472.465} C_VEL
LIN {X 0,Y 608.412,Z 269.505,A -85,B 0,C 180,E1 -474.572,E2 -474.572} C_VEL
LIN {X 0,Y 608.46,Z 269.504,A -85,B 0,C 180,E1 -477.204,E2 -477.204} C_VEL
LIN {X 0,Y 608.413,Z 269.508,A -85,B 0,C 180,E1 -479.963,E2 -479.963} C_VEL
LIN {X 0,Y 608.41,Z 269.505,A -85,B 0,C 180,E1 -482.515,E2 -482.515} C_VEL
LIN {X 0,Y 608.415,Z 269.508,A -85,B 0,C 180,E1 -484.901,E2 -484.901} C_VEL
LIN {X 0,Y 608.434,Z 269.506,A -85,B 0,C 180,E1 -487.748,E2 -487.748} C_VEL
LIN {X 0,Y 608.396,Z 269.507,A -85,B 0,C 180,E1 -490.323,E2 -490.323} C_VEL
LIN {X 0,Y 608.443,Z 269.508,A -85,B 0,C 180,E1 -492.959,E2 -492.959} C_VEL
LIN {X 0,Y 608.406,Z 269.507,A -85,B 0,C 180,E1 -495.74,E2 -495.74} C_VEL
LIN {X 0,Y 608.405,Z 269.506,A -85,B 0,C 180,E1 -497.934,E2 -497.934} C_VEL
LIN {X 0,Y 608.433,Z 269.508,A -85,B 0,C 180,E1 -500.705,E2 -500.705} C_VEL
LIN {X 0,Y 608.446,Z 269.509,A -85,B 0,C 180,E1 -503.084,E2 -503.084} C_VEL
LIN {X 0,Y 608.425,Z 269.505,A -85,B 0,C 180,E1 -505.528,E2 -505.528} C_VEL
LIN {X 0,Y 608.413,Z 269.505,A -85,B 0,C 180,E1 -507.903,E2 -507.903} C_VEL
LIN {X 0,Y 608.427,Z 269.506,A -85,B 0,C 180,E1 -510.218,E2 -510.218} C_VEL
LIN {X 0,Y 608.405,Z 269.508,A -85,B 0,C 180,E1 -513.224,E2 -513.224} C_VEL
LIN {X 0,Y 608.404,Z 269.506,A -85,B 0,C 180,E1 -515.427,E2 -515.427} C_VEL
LIN {X 0,Y 608.453,Z 269.506,A -85,B 0,C 180,E1 -518.308,E2 -518.308} C_VEL
LIN {X 0,Y 608.401,Z 269.507,A -85,B 0,C 180,E1 -521.3,E2 -521.3} C_VEL
LIN {X 0,Y 608.422,Z 269.506,A -85,B 0,C 180,E1 -523.905,E2 -523.905} C_VEL
LIN {X 0,Y 608.427,Z 269.509,A -85,B 0,C 180,E1 -526.643,E2 -526.643} C_VEL
LIN {X 0,Y 608.4,Z 269.507,A -85,B 0,C 180,E1 -529.349,E2 -529.349} C_VEL
LIN {X 0,Y 608.46,Z 269.506,A -85,B 0,C 180,E1 -532.033,E2 -532.033} C_VEL
LIN {X 0,Y 608.415,Z 269.507,A -85,B 0,C 180,E1 -534.698,E2 -534.698} C_VEL
LIN {X 0,Y 608.418,Z 269.505,A -85,B 0,C 180,E1 -537.352,E2 -537.352} C_VEL
LIN {X 0,Y 608.465,Z 269.509,A -85,B 0,C 180,E1 -540,E2 -540} C_VEL
LIN {X 0,Y 608.416,Z 269.506,A -85,B 0,C 180,E1 -542.648,E2 -542.648} C_VEL
LIN {X 0,Y 608.41,Z 269.507,A -85,B 0,C 180,E1 -545.302,E2 -545.302} C_VEL
LIN {X 0,Y 608.458,Z 269.507,A -85,B 0,C 180,E1 -547.967,E2 -547.967} C_VEL
LIN {X 0,Y 608.421,Z 269.507,A -85,B 0,C 180,E1 -549.417,E2 -549.417} C_VEL
LIN {X 0,Y 607.762,Z 269.594,A -85,B 0,C 180,E1 -549.97,E2 -549.97} C_VEL
LIN {X 0,Y 604.925,Z 269.946,A -85,B 0,C 180,E1 -550.867,E2 -550.867} C_VEL
LIN {X 0,Y 602.512,Z 270.248,A -85,B 0,C 180,E1 -551.588,E2 -551.588} C_VEL
LIN {X 0,Y 601.458,Z 270.375,A -85,B 0,C 180,E1 -552.144,E2 -552.144} C_VEL
LIN {X 0,Y 601.363,Z 270.385,A -85,B 0,C 180,E1 -552.333,E2 -552.333} C_VEL
LIN {X 0,Y 601.362,Z 270.384,A -85,B 0,C 180,E1 -554.899,E2 -554.899} C_VEL
LIN {X 0,Y 601.359,Z 270.392,A -85,B 0,C 180,E1 -557.69,E2 -557.69} C_VEL
LIN {X 0,Y 601.37,Z 270.388,A -85,B 0,C 180,E1 -559.811,E2 -559.811} C_VEL
LIN {X 0,Y 601.375,Z 270.385,A -85,B 0,C 180,E1 -561.961,E2 -561.961} C_VEL
LIN {X 0,Y 601.367,Z 270.385,A -85,B 0,C 180,E1 -564.88,E2 -564.88} C_VEL
LIN {X 0,Y 601.392,Z 270.39,A -85,B 0,C 180,E1 -567.361,E2 -567.361} C_VEL
LIN {X 0,Y 601.361,Z 270.384,A -85,B 0,C 180,E1 -570.168,E2 -570.168} C_VEL
LIN {X 0,Y 601.38,Z 270.384,A -85,B 0,C 180,E1 -572.711,E2 -572.711} C_VEL
LIN {X 0,Y 601.363,Z 270.393,A -85,B 0,C 180,E1 -575.109,E2 -575.109} C_VEL
LIN {X 0,Y 601.421,Z 270.381,A -85,B 0,C 180,E1 -577.42,E2 -577.42} C_VEL
LIN {X 0,Y 601.366,Z 270.383,A -85,B 0,C 180,E1 -579.999,E2 -579.999} C_VEL
LIN {X 0,Y 601.368,Z 270.388,A -85,B 0,C 180,E1 -582.674,E2 -582.674} C_VEL
LIN {X 0,Y 601.392,Z 270.382,A -85,B 0,C 180,E1 -585.48,E2 -585.48} C_VEL
LIN {X 0,Y 601.399,Z 270.382,A -85,B 0,C 180,E1 -588.41,E2 -588.41} C_VEL
LIN {X 0,Y 601.392,Z 270.389,A -85,B 0,C 180,E1 -590.873,E2 -590.873} C_VEL
LIN {X 0,Y 601.382,Z 270.382,A -85,B 0,C 180,E1 -593.417,E2 -593.417} C_VEL
LIN {X 0,Y 601.393,Z 270.381,A -85,B 0,C 180,E1 -596.07,E2 -596.07} C_VEL
LIN {X 0,Y 601.385,Z 270.383,A -85,B 0,C 180,E1 -599.057,E2 -599.057} C_VEL
LIN {X 0,Y 601.381,Z 270.381,A -85,B 0,C 180,E1 -601.371,E2 -601.371} C_VEL
LIN {X 0,Y 601.395,Z 270.384,A -85,B 0,C 180,E1 -604.136,E2 -604.136} C_VEL
LIN {X 0,Y 601.372,Z 270.388,A -85,B 0,C 180,E1 -606.588,E2 -606.588} C_VEL
LIN {X 0,Y 601.386,Z 270.382,A -85,B 0,C 180,E1 -609.477,E2 -609.477} C_VEL
LIN {X 0,Y 601.429,Z 270.545,A -85,B 0,C 180,E1 -610.236,E2 -610.236} C_VEL
LIN {X 0,Y 601.506,Z 281.936,A -85,B 0,C 180,E1 -612.315,E2 -612.315} C_VEL
LIN {X 0,Y 601.432,Z 297.548,A -85,B 0,C 180,E1 -615.104,E2 -615.104} C_VEL
LIN {X 0,Y 601.415,Z 313.161,A -85,B 0,C 180,E1 -617.858,E2 -617.858} C_VEL
LIN {X 0,Y 601.407,Z 323.541,A -85,B 0,C 180,E1 -619.65,E2 -619.65} C_VEL
LIN {X 0,Y 601.535,Z 325.212,A -85,B 0,C 180,E1 -619.716,E2 -619.716} C_VEL
LIN {X 0,Y 601.501,Z 400.297,A -85,B 0,C 180,E1 -620.628,E2 -620.628} C_VEL
LIN {X 0,Y 601.485,Z 410.811,A -85,B 0,C 180,E1 -620.861,E2 -620.861} C_VEL
LIN {X 0,Y 601.473,Z 422.546,A -85,B 0,C 180,E1 -621.263,E2 -621.263} C_VEL
LIN {X 0,Y 601.455,Z 432.935,A -85,B 0,C 180,E1 -621.771,E2 -621.771} C_VEL
LIN {X 0,Y 601.435,Z 441.116,A -85,B 0,C 180,E1 -622.277,E2 -622.277} C_VEL
LIN {X 0,Y 601.414,Z 448.877,A -85,B 0,C 180,E1 -622.868,E2 -622.868} C_VEL
LIN {X 0,Y 601.394,Z 456.707,A -85,B 0,C 180,E1 -623.598,E2 -623.598} C_VEL
LIN {X 0,Y 601.383,Z 464.116,A -85,B 0,C 180,E1 -624.467,E2 -624.467} C_VEL
LIN {X 0,Y 601.34,Z 469.729,A -85,B 0,C 180,E1 -625.307,E2 -625.307} C_VEL
LIN {X 0,Y 601.366,Z 474.944,A -85,B 0,C 180,E1 -626.315,E2 -626.315} C_VEL
LIN {X 0,Y 601.345,Z 477.633,A -85,B 0,C 180,E1 -626.985,E2 -626.985} C_VEL
LIN {X 0,Y 601.343,Z 480.571,A -85,B 0,C 180,E1 -627.991,E2 -627.991} C_VEL
LIN {X 0,Y 601.345,Z 481.871,A -85,B 0,C 180,E1 -628.661,E2 -628.661} C_VEL
LIN {X 0,Y 601.335,Z 482.692,A -85,B 0,C 180,E1 -629.33,E2 -629.33} C_VEL
LIN {X 0,Y 601.333,Z 482.996,A -85,B 0,C 180,E1 -630,E2 -630} C_VEL
LIN {X 0,Y 601.336,Z 482.734,A -85,B 0,C 180,E1 -630.67,E2 -630.67} C_VEL
LIN {X 0,Y 601.346,Z 481.997,A -85,B 0,C 180,E1 -631.339,E2 -631.339} C_VEL
LIN {X 0,Y 601.343,Z 480.786,A -85,B 0,C 180,E1 -632.009,E2 -632.009} C_VEL
LIN {X 0,Y 601.344,Z 477.941,A -85,B 0,C 180,E1 -633.015,E2 -633.015} C_VEL
LIN {X 0,Y 601.365,Z 475.35,A -85,B 0,C 180,E1 -633.685,E2 -633.685} C_VEL
LIN {X 0,Y 601.362,Z 470.243,A -85,B 0,C 180,E1 -634.692,E2 -634.692} C_VEL
LIN {X 0,Y 601.384,Z 464.747,A -85,B 0,C 180,E1 -635.532,E2 -635.532} C_VEL
LIN {X 0,Y 601.394,Z 456.588,A -85,B 0,C 180,E1 -636.504,E2 -636.504} C_VEL
LIN {X 0,Y 601.413,Z 448.944,A -85,B 0,C 180,E1 -637.217,E2 -637.217} C_VEL
LIN {X 0,Y 601.412,Z 441.195,A -85,B 0,C 180,E1 -637.807,E2 -637.807} C_VEL
LIN {X 0,Y 601.447,Z 433.03,A -85,B 0,C 180,E1 -638.314,E2 -638.314} C_VEL
LIN {X 0,Y 601.461,Z 422.663,A -85,B 0,C 180,E1 -638.822,E2 -638.822} C_VEL
LIN {X 0,Y 601.491,Z 411.015,A -85,B 0,C 180,E1 -639.224,E2 -639.224} C_VEL
LIN {X 0,Y 601.512,Z 400.616,A -85,B 0,C 180,E1 -639.457,E2 -639.457} C_VEL
LIN {X 0,Y 601.553,Z 352.361,A -85,B 0,C 180,E1 -640.05,E2 -640.05} C_VEL
LIN {X 0,Y 601.461,Z 324.339,A -85,B 0,C 180,E1 -640.392,E2 -640.392} C_VEL
LIN {X 0,Y 601.393,Z 323.245,A -85,B 0,C 180,E1 -640.478,E2 -640.478} C_VEL
LIN {X 0,Y 601.397,Z 307.817,A -85,B 0,C 180,E1 -643.172,E2 -643.172} C_VEL
LIN {X 0,Y 601.439,Z 292.198,A -85,B 0,C 180,E1 -645.938,E2 -645.938} C_VEL
LIN {X 0,Y 601.528,Z 275.981,A -85,B 0,C 180,E1 -648.849,E2 -648.849} C_VEL
LIN {X 0,Y 601.419,Z 270.442,A -85,B 0,C 180,E1 -649.897,E2 -649.897} C_VEL
LIN {X 0,Y 601.398,Z 270.376,A -85,B 0,C 180,E1 -652.683,E2 -652.683} C_VEL
LIN {X 0,Y 601.433,Z 270.385,A -85,B 0,C 180,E1 -655.617,E2 -655.617} C_VEL
LIN {X 0,Y 601.359,Z 270.389,A -85,B 0,C 180,E1 -657.87,E2 -657.87} C_VEL
LIN {X 0,Y 601.394,Z 270.381,A -85,B 0,C 180,E1 -660.165,E2 -660.165} C_VEL
LIN {X 0,Y 601.388,Z 270.381,A -85,B 0,C 180,E1 -662.71,E2 -662.71} C_VEL
LIN {X 0,Y 601.371,Z 270.388,A -85,B 0,C 180,E1 -665.108,E2 -665.108} C_VEL
LIN {X 0,Y 601.427,Z 270.384,A -85,B 0,C 180,E1 -667.419,E2 -667.419} C_VEL
LIN {X 0,Y 601.371,Z 270.383,A -85,B 0,C 180,E1 -669.997,E2 -669.997} C_VEL
LIN {X 0,Y 601.37,Z 270.385,A -85,B 0,C 180,E1 -672.673,E2 -672.673} C_VEL
LIN {X 0,Y 601.392,Z 270.384,A -85,B 0,C 180,E1 -675.479,E2 -675.479} C_VEL
LIN {X 0,Y 601.4,Z 270.38,A -85,B 0,C 180,E1 -678.408,E2 -678.408} C_VEL
LIN {X 0,Y 601.396,Z 270.387,A -85,B 0,C 180,E1 -680.872,E2 -680.872} C_VEL
LIN {X 0,Y 601.39,Z 270.383,A -85,B 0,C 180,E1 -683.416,E2 -683.416} C_VEL
LIN {X 0,Y 601.389,Z 270.38,A -85,B 0,C 180,E1 -686.069,E2 -686.069} C_VEL
LIN {X 0,Y 601.404,Z 270.384,A -85,B 0,C 180,E1 -688.546,E2 -688.546} C_VEL
LIN {X 0,Y 601.382,Z 270.382,A -85,B 0,C 180,E1 -691.37,E2 -691.37} C_VEL
LIN {X 0,Y 601.365,Z 270.383,A -85,B 0,C 180,E1 -693.634,E2 -693.634} C_VEL
LIN {X 0,Y 601.387,Z 270.381,A -85,B 0,C 180,E1 -695.857,E2 -695.857} C_VEL
LIN {X 0,Y 601.385,Z 270.387,A -85,B 0,C 180,E1 -698.76,E2 -698.76} C_VEL
LIN {X 0,Y 601.35,Z 270.385,A -85,B 0,C 180,E1 -701.606,E2 -701.606} C_VEL
LIN {X 0,Y 601.382,Z 270.392,A -85,B 0,C 180,E1 -704.408,E2 -704.408} C_VEL
LIN {X 0,Y 601.348,Z 270.385,A -85,B 0,C 180,E1 -707.17,E2 -707.17} C_VEL
LIN {X 0,Y 601.413,Z 270.381,A -85,B 0,C 180,E1 -709.905,E2 -709.905} C_VEL
LIN {X 0,Y 601.381,Z 270.385,A -85,B 0,C 180,E1 -712.614,E2 -712.614} C_VEL
LIN {X 0,Y 601.387,Z 270.383,A -85,B 0,C 180,E1 -714.635,E2 -714.635} C_VEL
LIN {X 0,Y 601.386,Z 270.381,A -85,B 0,C 180,E1 -717.321,E2 -717.321} C_VEL
LIN {X 0,Y 601.433,Z 270.385,A -85,B 0,C 180,E1 -720,E2 -720} C_VEL
LIN {X 0,Y 601.384,Z 270.381,A -85,B 0,C 180,E1 -722.679,E2 -722.679} C_VEL
LIN {X 0,Y 601.382,Z 270.383,A -85,B 0,C 180,E1 -725.364,E2 -725.364} C_VEL
LIN {X 0,Y 601.416,Z 270.383,A -85,B 0,C 180,E1 -728.061,E2 -728.061} C_VEL
LIN {X 0,Y 601.365,Z 270.384,A -85,B 0,C 180,E1 -730.989,E2 -730.989} C_VEL
LIN {X 0,Y 601.377,Z 270.389,A -85,B 0,C 180,E1 -733.517,E2 -733.517} C_VEL
LIN {X 0,Y 601.378,Z 270.383,A -85,B 0,C 180,E1 -736.289,E2 -736.289} C_VEL
LIN {X 0,Y 601.39,Z 270.383,A -85,B 0,C 180,E1 -739.1,E2 -739.1} C_VEL
LIN {X 0,Y 601.375,Z 270.384,A -85,B 0,C 180,E1 -741.961,E2 -741.961} C_VEL
LIN {X 0,Y 601.367,Z 270.385,A -85,B 0,C 180,E1 -744.88,E2 -744.88} C_VEL
LIN {X 0,Y 601.392,Z 270.39,A -85,B 0,C 180,E1 -747.361,E2 -747.361} C_VEL
LIN {X 0,Y 601.36,Z 270.384,A -85,B 0,C 180,E1 -750.168,E2 -750.168} C_VEL
LIN {X 0,Y 601.381,Z 270.384,A -85,B 0,C 180,E1 -752.711,E2 -752.711} C_VEL
LIN {X 0,Y 601.366,Z 270.393,A -85,B 0,C 180,E1 -755.11,E2 -755.11} C_VEL
LIN {X 0,Y 601.421,Z 270.381,A -85,B 0,C 180,E1 -757.42,E2 -757.42} C_VEL
LIN {X 0,Y 601.366,Z 270.383,A -85,B 0,C 180,E1 -759.999,E2 -759.999} C_VEL
LIN {X 0,Y 601.371,Z 270.388,A -85,B 0,C 180,E1 -762.674,E2 -762.674} C_VEL
LIN {X 0,Y 601.391,Z 270.381,A -85,B 0,C 180,E1 -765.48,E2 -765.48} C_VEL
LIN {X 0,Y 601.401,Z 270.382,A -85,B 0,C 180,E1 -768.409,E2 -768.409} C_VEL
LIN {X 0,Y 601.393,Z 270.388,A -85,B 0,C 180,E1 -770.873,E2 -770.873} C_VEL
LIN {X 0,Y 601.383,Z 270.382,A -85,B 0,C 180,E1 -773.417,E2 -773.417} C_VEL
LIN {X 0,Y 601.405,Z 270.38,A -85,B 0,C 180,E1 -776.068,E2 -776.068} C_VEL
LIN {X 0,Y 601.385,Z 270.383,A -85,B 0,C 180,E1 -779.057,E2 -779.057} C_VEL
LIN {X 0,Y 601.384,Z 270.381,A -85,B 0,C 180,E1 -781.371,E2 -781.371} C_VEL
LIN {X 0,Y 601.397,Z 270.385,A -85,B 0,C 180,E1 -784.136,E2 -784.136} C_VEL
LIN {X 0,Y 601.375,Z 270.387,A -85,B 0,C 180,E1 -786.588,E2 -786.588} C_VEL
LIN {X 0,Y 601.39,Z 270.382,A -85,B 0,C 180,E1 -789.477,E2 -789.477} C_VEL
LIN {X 0,Y 601.419,Z 270.547,A -85,B 0,C 180,E1 -790.192,E2 -790.192} C_VEL
LIN {X 0,Y 601.49,Z 282.186,A -85,B 0,C 180,E1 -792.315,E2 -792.315} C_VEL
LIN {X 0,Y 601.431,Z 297.802,A -85,B 0,C 180,E1 -795.103,E2 -795.103} C_VEL
LIN {X 0,Y 601.414,Z 313.418,A -85,B 0,C 180,E1 -797.858,E2 -797.858} C_VEL
LIN {X 0,Y 601.401,Z 323.567,A -85,B 0,C 180,E1 -799.607,E2 -799.607} C_VEL
LIN {X 0,Y 601.528,Z 325.352,A -85,B 0,C 180,E1 -799.673,E2 -799.673} C_VEL
LIN {X 0,Y 601.518,Z 399.156,A -85,B 0,C 180,E1 -800.565,E2 -800.565} C_VEL
LIN {X 0,Y 601.511,Z 408.422,A -85,B 0,C 180,E1 -800.755,E2 -800.755} C_VEL
LIN {X 0,Y 601.472,Z 416.895,A -85,B 0,C 180,E1 -801.009,E2 -801.009} C_VEL
LIN {X 0,Y 601.481,Z 425.396,A -85,B 0,C 180,E1 -801.348,E2 -801.348} C_VEL
LIN {X 0,Y 601.454,Z 433.725,A -85,B 0,C 180,E1 -801.771,E2 -801.771} C_VEL
LIN {X 0,Y 601.432,Z 441.764,A -85,B 0,C 180,E1 -802.277,E2 -802.277} C_VEL
LIN {X 0,Y 601.414,Z 449.417,A -85,B 0,C 180,E1 -802.868,E2 -802.868} C_VEL
LIN {X 0,Y 601.393,Z 457.152,A -85,B 0,C 180,E1 -803.597,E2 -803.597} C_VEL
LIN {X 0,Y 601.383,Z 464.432,A -85,B 0,C 180,E1 -804.467,E2 -804.467} C_VEL
LIN {X 0,Y 601.341,Z 469.986,A -85,B 0,C 180,E1 -805.307,E2 -805.307} C_VEL
LIN {X 0,Y 601.364,Z 475.147,A -85,B 0,C 180,E1 -806.315,E2 -806.315} C_VEL
LIN {X 0,Y 601.342,Z 477.787,A -85,B 0,C 180,E1 -806.985,E2 -806.985} C_VEL
LIN {X 0,Y 601.343,Z 480.679,A -85,B 0,C 180,E1 -807.991,E2 -807.991} C_VEL
LIN {X 0,Y 601.345,Z 481.934,A -85,B 0,C 180,E1 -808.661,E2 -808.661} C_VEL
LIN {X 0,Y 601.335,Z 482.713,A -85,B 0,C 180,E1 -809.33,E2 -809.33} C_VEL
LIN {X 0,Y 601.332,Z 483,A -85,B 0,C 180,E1 -810,E2 -810} C_VEL
LIN {X 0,Y 601.335,Z 482.713,A -85,B 0,C 180,E1 -810.67,E2 -810.67} C_VEL
LIN {X 0,Y 601.345,Z 481.934,A -85,B 0,C 180,E1 -811.339,E2 -811.339} C_VEL
LIN {X 0,Y 601.343,Z 480.679,A -85,B 0,C 180,E1 -812.009,E2 -812.009} C_VEL
LIN {X 0,Y 601.342,Z 477.787,A -85,B 0,C 180,E1 -813.015,E2 -813.015} C_VEL
LIN {X 0,Y 601.364,Z 475.147,A -85,B 0,C 180,E1 -813.685,E2 -813.685} C_VEL
LIN {X 0,Y 601.341,Z 469.986,A -85,B 0,C 180,E1 -814.693,E2 -814.693} C_VEL
LIN {X 0,Y 601.383,Z 464.431,A -85,B 0,C 180,E1 -815.533,E2 -815.533} C_VEL
LIN {X 0,Y 601.393,Z 457.152,A -85,B 0,C 180,E1 -816.403,E2 -816.403} C_VEL
LIN {X 0,Y 601.414,Z 449.418,A -85,B 0,C 180,E1 -817.132,E2 -817.132} C_VEL
LIN {X 0,Y 601.432,Z 441.765,A -85,B 0,C 180,E1 -817.723,E2 -817.723} C_VEL
LIN {X 0,Y 601.454,Z 433.726,A -85,B 0,C 180,E1 -818.229,E2 -818.229} C_VEL
LIN {X 0,Y 601.481,Z 425.397,A -85,B 0,C 180,E1 -818.652,E2 -818.652} C_VEL
LIN {X 0,Y 601.472,Z 416.896,A -85,B 0,C 180,E1 -818.991,E2 -818.991} C_VEL
LIN {X 0,Y 601.498,Z 407.593,A -85,B 0,C 180,E1 -819.266,E2 -819.266} C_VEL
LIN {X 0,Y 601.528,Z 396.56,A -85,B 0,C 180,E1 -819.478,E2 -819.478} C_VEL
LIN {X 0,Y 601.452,Z 324.257,A -85,B 0,C 180,E1 -820.35,E2 -820.35} C_VEL
LIN {X 0,Y 601.386,Z 323.229,A -85,B 0,C 180,E1 -820.436,E2 -820.436} C_VEL
LIN {X 0,Y 601.39,Z 309.514,A -85,B 0,C 180,E1 -822.828,E2 -822.828} C_VEL
LIN {X 0,Y 601.455,Z 293.898,A -85,B 0,C 180,E1 -825.59,E2 -825.59} C_VEL
LIN {X 0,Y 601.506,Z 277.006,A -85,B 0,C 180,E1 -828.619,E2 -828.619} C_VEL
LIN {X 0,Y 601.425,Z 270.443,A -85,B 0,C 180,E1 -829.853,E2 -829.853} C_VEL
LIN {X 0,Y 601.372,Z 270.379,A -85,B 0,C 180,E1 -832.684,E2 -832.684} C_VEL
LIN {X 0,Y 601.43,Z 270.385,A -85,B 0,C 180,E1 -835.617,E2 -835.617} C_VEL
LIN {X 0,Y 601.356,Z 270.389,A -85,B 0,C 180,E1 -837.87,E2 -837.87} C_VEL
LIN {X 0,Y 601.368,Z 270.384,A -85,B 0,C 180,E1 -840.167,E2 -840.167} C_VEL
LIN {X 0,Y 601.386,Z 270.381,A -85,B 0,C 180,E1 -842.71,E2 -842.71} C_VEL
LIN {X 0,Y 601.368,Z 270.389,A -85,B 0,C 180,E1 -845.108,E2 -845.108} C_VEL
LIN {X 0,Y 601.425,Z 270.384,A -85,B 0,C 180,E1 -847.419,E2 -847.419} C_VEL
LIN {X 0,Y 601.369,Z 270.383,A -85,B 0,C 180,E1 -849.997,E2 -849.997} C_VEL
LIN {X 0,Y 601.368,Z 270.385,A -85,B 0,C 180,E1 -852.673,E2 -852.673} C_VEL
LIN {X 0,Y 601.391,Z 270.384,A -85,B 0,C 180,E1 -855.479,E2 -855.479} C_VEL
LIN {X 0,Y 601.398,Z 270.38,A -85,B 0,C 180,E1 -858.408,E2 -858.408} C_VEL
LIN {X 0,Y 601.394,Z 270.388,A -85,B 0,C 180,E1 -860.872,E2 -860.872} C_VEL
LIN {X 0,Y 601.387,Z 270.383,A -85,B 0,C 180,E1 -863.416,E2 -863.416} C_VEL
LIN {X 0,Y 601.388,Z 270.381,A -85,B 0,C 180,E1 -866.069,E2 -866.069} C_VEL
LIN {X 0,Y 601.384,Z 270.386,A -85,B 0,C 180,E1 -869.056,E2 -869.056} C_VEL
LIN {X 0,Y 601.38,Z 270.382,A -85,B 0,C 180,E1 -871.371,E2 -871.371} C_VEL
LIN {X 0,Y 601.364,Z 270.383,A -85,B 0,C 180,E1 -873.634,E2 -873.634} C_VEL
LIN {X 0,Y 601.385,Z 270.381,A -85,B 0,C 180,E1 -875.857,E2 -875.857} C_VEL
LIN {X 0,Y 601.385,Z 270.387,A -85,B 0,C 180,E1 -878.76,E2 -878.76} C_VEL
LIN {X 0,Y 601.35,Z 270.385,A -85,B 0,C 180,E1 -881.606,E2 -881.606} C_VEL
LIN {X 0,Y 601.381,Z 270.392,A -85,B 0,C 180,E1 -884.408,E2 -884.408} C_VEL
LIN {X 0,Y 601.38,Z 270.389,A -85,B 0,C 180,E1 -886.483,E2 -886.483} C_VEL
LIN {X 0,Y 601.348,Z 270.385,A -85,B 0,C 180,E1 -889.223,E2 -889.223} C_VEL
LIN {X 0,Y 601.418,Z 270.382,A -85,B 0,C 180,E1 -891.939,E2 -891.939} C_VEL
LIN {X 0,Y 601.387,Z 270.383,A -85,B 0,C 180,E1 -894.636,E2 -894.636} C_VEL
LIN {X 0,Y 601.386,Z 270.381,A -85,B 0,C 180,E1 -897.321,E2 -897.321} C_VEL
LIN {X 0,Y 601.433,Z 270.385,A -85,B 0,C 180,E1 -900,E2 -900} C_VEL
LIN {X 0,Y 601.384,Z 270.381,A -85,B 0,C 180,E1 -902.679,E2 -902.679} C_VEL
LIN {X 0,Y 601.383,Z 270.383,A -85,B 0,C 180,E1 -905.365,E2 -905.365} C_VEL
LIN {X 0,Y 601.416,Z 270.383,A -85,B 0,C 180,E1 -908.061,E2 -908.061} C_VEL
LIN {X 0,Y 601.364,Z 270.384,A -85,B 0,C 180,E1 -910.989,E2 -910.989} C_VEL
LIN {X 0,Y 601.363,Z 270.385,A -85,B 0,C 180,E1 -912.333,E2 -912.333} C_VEL
LIN {X 0,Y 600.672,Z 270.471,A -85,B 0,C 180,E1 -912.892,E2 -912.892} C_VEL
LIN {X 0,Y 597.818,Z 270.833,A -85,B 0,C 180,E1 -913.8,E2 -913.8} C_VEL
LIN {X 0,Y 595.423,Z 271.128,A -85,B 0,C 180,E1 -914.53,E2 -914.53} C_VEL
LIN {X 0,Y 594.396,Z 271.253,A -85,B 0,C 180,E1 -915.094,E2 -915.094} C_VEL
LIN {X 0,Y 594.312,Z 271.264,A -85,B 0,C 180,E1 -915.285,E2 -915.285} C_VEL
LIN {X 0,Y 594.308,Z 271.267,A -85,B 0,C 180,E1 -917.907,E2 -917.907} C_VEL
LIN {X 0,Y 594.358,Z 271.256,A -85,B 0,C 180,E1 -920.777,E2 -920.777} C_VEL
LIN {X 0,Y 594.331,Z 271.265,A -85,B 0,C 180,E1 -923.707,E2 -923.707} C_VEL
LIN {X 0,Y 594.338,Z 271.26,A -85,B 0,C 180,E1 -926.016,E2 -926.016} C_VEL
LIN {X 0,Y 594.302,Z 271.263,A -85,B 0,C 180,E1 -928.231,E2 -928.231} C_VEL
LIN {X 0,Y 594.341,Z 271.259,A -85,B 0,C 180,E1 -930.562,E2 -930.562} C_VEL
LIN {X 0,Y 594.36,Z 271.261,A -85,B 0,C 180,E1 -932.951,E2 -932.951} C_VEL
LIN {X 0,Y 594.307,Z 271.268,A -85,B 0,C 180,E1 -935.412,E2 -935.412} C_VEL
LIN {X 0,Y 594.339,Z 271.258,A -85,B 0,C 180,E1 -937.944,E2 -937.944} C_VEL
LIN {X 0,Y 594.352,Z 271.263,A -85,B 0,C 180,E1 -940.821,E2 -940.821} C_VEL
LIN {X 0,Y 594.334,Z 271.259,A -85,B 0,C 180,E1 -943.837,E2 -943.837} C_VEL
LIN {X 0,Y 594.335,Z 271.266,A -85,B 0,C 180,E1 -946.699,E2 -946.699} C_VEL
LIN {X 0,Y 594.333,Z 271.26,A -85,B 0,C 180,E1 -949.431,E2 -949.431} C_VEL
LIN {X 0,Y 594.371,Z 271.259,A -85,B 0,C 180,E1 -952.394,E2 -952.394} C_VEL
LIN {X 0,Y 594.349,Z 271.258,A -85,B 0,C 180,E1 -955.419,E2 -955.419} C_VEL
LIN {X 0,Y 594.332,Z 271.26,A -85,B 0,C 180,E1 -957.852,E2 -957.852} C_VEL
LIN {X 0,Y 594.333,Z 271.264,A -85,B 0,C 180,E1 -960.222,E2 -960.222} C_VEL
LIN {X 0,Y 594.35,Z 271.257,A -85,B 0,C 180,E1 -963.299,E2 -963.299} C_VEL
LIN {X 0,Y 594.331,Z 271.26,A -85,B 0,C 180,E1 -965.579,E2 -965.579} C_VEL
LIN {X 0,Y 594.342,Z 271.267,A -85,B 0,C 180,E1 -968.496,E2 -968.496} C_VEL
LIN {X 0,Y 594.372,Z 271.41,A -85,B 0,C 180,E1 -970.149,E2 -970.149} C_VEL
LIN {X 0,Y 594.477,Z 279.988,A -85,B 0,C 180,E1 -971.743,E2 -971.743} C_VEL
LIN {X 0,Y 594.408,Z 295.6,A -85,B 0,C 180,E1 -974.572,E2 -974.572} C_VEL
LIN {X 0,Y 594.342,Z 311.213,A -85,B 0,C 180,E1 -977.364,E2 -977.364} C_VEL
LIN {X 0,Y 594.319,Z 323.546,A -85,B 0,C 180,E1 -979.525,E2 -979.525} C_VEL
LIN {X 0,Y 594.526,Z 325.242,A -85,B 0,C 180,E1 -979.593,E2 -979.593} C_VEL
LIN {X 0,Y 594.519,Z 400.328,A -85,B 0,C 180,E1 -980.517,E2 -980.517} C_VEL
LIN {X 0,Y 594.483,Z 410.833,A -85,B 0,C 180,E1 -980.752,E2 -980.752} C_VEL
LIN {X 0,Y 594.458,Z 422.555,A -85,B 0,C 180,E1 -981.159,E2 -981.159} C_VEL
LIN {X 0,Y 594.431,Z 432.947,A -85,B 0,C 180,E1 -981.673,E2 -981.673} C_VEL
LIN {X 0,Y 594.371,Z 441.127,A -85,B 0,C 180,E1 -982.185,E2 -982.185} C_VEL
LIN {X 0,Y 594.356,Z 448.885,A -85,B 0,C 180,E1 -982.783,E2 -982.783} C_VEL
LIN {X 0,Y 594.345,Z 456.712,A -85,B 0,C 180,E1 -983.522,E2 -983.522} C_VEL
LIN {X 0,Y 594.308,Z 464.12,A -85,B 0,C 180,E1 -984.401,E2 -984.401} C_VEL
LIN {X 0,Y 594.255,Z 469.732,A -85,B 0,C 180,E1 -985.251,E2 -985.251} C_VEL
LIN {X 0,Y 594.287,Z 474.946,A -85,B 0,C 180,E1 -986.271,E2 -986.271} C_VEL
LIN {X 0,Y 594.248,Z 477.635,A -85,B 0,C 180,E1 -986.949,E2 -986.949} C_VEL
LIN {X 0,Y 594.242,Z 480.573,A -85,B 0,C 180,E1 -987.967,E2 -987.967} C_VEL
LIN {X 0,Y 594.244,Z 481.873,A -85,B 0,C 180,E1 -988.645,E2 -988.645} C_VEL
LIN {X 0,Y 594.235,Z 482.691,A -85,B 0,C 180,E1 -989.322,E2 -989.322} C_VEL
LIN {X 0,Y 594.234,Z 482.996,A -85,B 0,C 180,E1 -990,E2 -990} C_VEL
LIN {X 0,Y 594.236,Z 482.734,A -85,B 0,C 180,E1 -990.678,E2 -990.678} C_VEL
LIN {X 0,Y 594.246,Z 481.998,A -85,B 0,C 180,E1 -991.355,E2 -991.355} C_VEL
LIN {X 0,Y 594.242,Z 480.786,A -85,B 0,C 180,E1 -992.033,E2 -992.033} C_VEL
LIN {X 0,Y 594.247,Z 477.939,A -85,B 0,C 180,E1 -993.051,E2 -993.051} C_VEL
LIN {X 0,Y 594.286,Z 475.348,A -85,B 0,C 180,E1 -993.729,E2 -993.729} C_VEL
LIN {X 0,Y 594.265,Z 470.24,A -85,B 0,C 180,E1 -994.749,E2 -994.749} C_VEL
LIN {X 0,Y 594.31,Z 464.744,A -85,B 0,C 180,E1 -995.599,E2 -995.599} C_VEL
LIN {X 0,Y 594.342,Z 457.617,A -85,B 0,C 180,E1 -996.476,E2 -996.476} C_VEL
LIN {X 0,Y 594.354,Z 448.938,A -85,B 0,C 180,E1 -997.303,E2 -997.303} C_VEL
LIN {X 0,Y 594.378,Z 441.19,A -85,B 0,C 180,E1 -997.9,E2 -997.9} C_VEL
LIN {X 0,Y 594.42,Z 433.024,A -85,B 0,C 180,E1 -998.413,E2 -998.413} C_VEL
LIN {X 0,Y 594.46,Z 422.648,A -85,B 0,C 180,E1 -998.926,E2 -998.926} C_VEL
LIN {X 0,Y 594.49,Z 410.994,A -85,B 0,C 180,E1 -999.333,E2 -999.333} C_VEL
LIN {X 0,Y 594.53,Z 400.583,A -85,B 0,C 180,E1 -999.569,E2 -999.569} C_VEL
LIN {X 0,Y 594.577,Z 352.316,A -85,B 0,C 180,E1 -1000.169,E2 -1000.169} C_VEL
LIN {X 0,Y 594.4,Z 324.304,A -85,B 0,C 180,E1 -1000.517,E2 -1000.517} C_VEL
LIN {X 0,Y 594.309,Z 322.962,A -85,B 0,C 180,E1 -1000.648,E2 -1000.648} C_VEL
LIN {X 0,Y 594.362,Z 307.814,A -85,B 0,C 180,E1 -1003.331,E2 -1003.331} C_VEL
LIN {X 0,Y 594.411,Z 292.195,A -85,B 0,C 180,E1 -1006.132,E2 -1006.132} C_VEL
LIN {X 0,Y 594.529,Z 276.578,A -85,B 0,C 180,E1 -1008.97,E2 -1008.97} C_VEL
LIN {X 0,Y 594.381,Z 271.347,A -85,B 0,C 180,E1 -1009.963,E2 -1009.963} C_VEL
LIN {X 0,Y 594.345,Z 271.254,A -85,B 0,C 180,E1 -1012.967,E2 -1012.967} C_VEL
LIN {X 0,Y 594.361,Z 271.26,A -85,B 0,C 180,E1 -1015.944,E2 -1015.944} C_VEL
LIN {X 0,Y 594.367,Z 271.256,A -85,B 0,C 180,E1 -1018.955,E2 -1018.955} C_VEL
LIN {X 0,Y 594.364,Z 271.263,A -85,B 0,C 180,E1 -1021.64,E2 -1021.64} C_VEL
LIN {X 0,Y 594.355,Z 271.256,A -85,B 0,C 180,E1 -1024.581,E2 -1024.581} C_VEL
LIN {X 0,Y 594.377,Z 271.259,A -85,B 0,C 180,E1 -1027.607,E2 -1027.607} C_VEL
LIN {X 0,Y 594.336,Z 271.26,A -85,B 0,C 180,E1 -1030.569,E2 -1030.569} C_VEL
LIN {X 0,Y 594.338,Z 271.267,A -85,B 0,C 180,E1 -1033.301,E2 -1033.301} C_VEL
LIN {X 0,Y 594.334,Z 271.259,A -85,B 0,C 180,E1 -1036.163,E2 -1036.163} C_VEL
LIN {X 0,Y 594.364,Z 271.263,A -85,B 0,C 180,E1 -1039.178,E2 -1039.178} C_VEL
LIN {X 0,Y 594.356,Z 271.256,A -85,B 0,C 180,E1 -1042.057,E2 -1042.057} C_VEL
LIN {X 0,Y 594.312,Z 271.268,A -85,B 0,C 180,E1 -1044.68,E2 -1044.68} C_VEL
LIN {X 0,Y 594.361,Z 271.262,A -85,B 0,C 180,E1 -1047.089,E2 -1047.089} C_VEL
LIN {X 0,Y 594.337,Z 271.259,A -85,B 0,C 180,E1 -1049.678,E2 -1049.678} C_VEL
LIN {X 0,Y 594.308,Z 271.262,A -85,B 0,C 180,E1 -1051.769,E2 -1051.769} C_VEL
LIN {X 0,Y 594.345,Z 271.259,A -85,B 0,C 180,E1 -1054.054,E2 -1054.054} C_VEL
LIN {X 0,Y 594.325,Z 271.263,A -85,B 0,C 180,E1 -1057.031,E2 -1057.031} C_VEL
LIN {X 0,Y 594.362,Z 271.256,A -85,B 0,C 180,E1 -1059.223,E2 -1059.223} C_VEL
LIN {X 0,Y 594.312,Z 271.266,A -85,B 0,C 180,E1 -1062.094,E2 -1062.094} C_VEL
LIN {X 0,Y 594.324,Z 271.263,A -85,B 0,C 180,E1 -1064.921,E2 -1064.921} C_VEL
LIN {X 0,Y 594.353,Z 271.258,A -85,B 0,C 180,E1 -1067.711,E2 -1067.711} C_VEL
LIN {X 0,Y 594.335,Z 271.265,A -85,B 0,C 180,E1 -1070.471,E2 -1070.471} C_VEL
LIN {X 0,Y 594.326,Z 271.26,A -85,B 0,C 180,E1 -1073.209,E2 -1073.209} C_VEL
LIN {X 0,Y 594.339,Z 271.265,A -85,B 0,C 180,E1 -1075.931,E2 -1075.931} C_VEL
LIN {X 0,Y 594.329,Z 271.261,A -85,B 0,C 180,E1 -1078.645,E2 -1078.645} C_VEL
LIN {X 0,Y 594.311,Z 271.263,A -85,B 0,C 180,E1 -1080.677,E2 -1080.677} C_VEL
LIN {X 0,Y 594.352,Z 271.257,A -85,B 0,C 180,E1 -1082.711,E2 -1082.711} C_VEL
LIN {X 0,Y 594.353,Z 271.26,A -85,B 0,C 180,E1 -1085.428,E2 -1085.428} C_VEL
LIN {X 0,Y 594.358,Z 271.261,A -85,B 0,C 180,E1 -1088.157,E2 -1088.157} C_VEL
LIN {X 0,Y 594.332,Z 271.26,A -85,B 0,C 180,E1 -1091.052,E2 -1091.052} C_VEL
LIN {X 0,Y 594.344,Z 271.268,A -85,B 0,C 180,E1 -1093.68,E2 -1093.68} C_VEL
LIN {X 0,Y 594.307,Z 271.262,A -85,B 0,C 180,E1 -1096.695,E2 -1096.695} C_VEL
LIN {X 0,Y 594.341,Z 271.265,A -85,B 0,C 180,E1 -1099.335,E2 -1099.335} C_VEL
LIN {X 0,Y 594.339,Z 271.269,A -85,B 0,C 180,E1 -1101.504,E2 -1101.504} C_VEL
LIN {X 0,Y 594.329,Z 271.259,A -85,B 0,C 180,E1 -1104.449,E2 -1104.449} C_VEL
LIN {X 0,Y 594.345,Z 271.259,A -85,B 0,C 180,E1 -1106.701,E2 -1106.701} C_VEL
LIN {X 0,Y 594.324,Z 271.263,A -85,B 0,C 180,E1 -1109.779,E2 -1109.779} C_VEL
LIN {X 0,Y 594.328,Z 271.26,A -85,B 0,C 180,E1 -1112.149,E2 -1112.149} C_VEL
LIN {X 0,Y 594.349,Z 271.259,A -85,B 0,C 180,E1 -1114.582,E2 -1114.582} C_VEL
LIN {X 0,Y 594.371,Z 271.257,A -85,B 0,C 180,E1 -1117.608,E2 -1117.608} C_VEL
LIN {X 0,Y 594.333,Z 271.262,A -85,B 0,C 180,E1 -1120.57,E2 -1120.57} C_VEL
LIN {X 0,Y 594.335,Z 271.263,A -85,B 0,C 180,E1 -1123.302,E2 -1123.302} C_VEL
LIN {X 0,Y 594.335,Z 271.26,A -85,B 0,C 180,E1 -1126.164,E2 -1126.164} C_VEL
LIN {X 0,Y 594.354,Z 271.26,A -85,B 0,C 180,E1 -1129.181,E2 -1129.181} C_VEL
LIN {X 0,Y 594.343,Z 271.259,A -85,B 0,C 180,E1 -1132.057,E2 -1132.057} C_VEL
LIN {X 0,Y 594.314,Z 271.271,A -85,B 0,C 180,E1 -1134.681,E2 -1134.681} C_VEL
LIN {X 0,Y 594.364,Z 271.258,A -85,B 0,C 180,E1 -1137.091,E2 -1137.091} C_VEL
LIN {X 0,Y 594.342,Z 271.258,A -85,B 0,C 180,E1 -1139.679,E2 -1139.679} C_VEL
LIN {X 0,Y 594.311,Z 271.263,A -85,B 0,C 180,E1 -1141.77,E2 -1141.77} C_VEL
LIN {X 0,Y 594.355,Z 271.261,A -85,B 0,C 180,E1 -1144.056,E2 -1144.056} C_VEL
LIN {X 0,Y 594.333,Z 271.258,A -85,B 0,C 180,E1 -1147.032,E2 -1147.032} C_VEL
LIN {X 0,Y 594.392,Z 271.347,A -85,B 0,C 180,E1 -1150.083,E2 -1150.083} C_VEL
LIN {X 0,Y 594.473,Z 280.234,A -85,B 0,C 180,E1 -1151.743,E2 -1151.743} C_VEL
LIN {X 0,Y 594.407,Z 295.85,A -85,B 0,C 180,E1 -1154.572,E2 -1154.572} C_VEL
LIN {X 0,Y 594.34,Z 311.466,A -85,B 0,C 180,E1 -1157.364,E2 -1157.364} C_VEL
LIN {X 0,Y 594.331,Z 323.567,A -85,B 0,C 180,E1 -1159.482,E2 -1159.482} C_VEL
LIN {X 0,Y 594.519,Z 325.352,A -85,B 0,C 180,E1 -1159.55,E2 -1159.55} C_VEL
LIN {X 0,Y 594.535,Z 399.155,A -85,B 0,C 180,E1 -1160.453,E2 -1160.453} C_VEL
LIN {X 0,Y 594.511,Z 408.422,A -85,B 0,C 180,E1 -1160.646,E2 -1160.646} C_VEL
LIN {X 0,Y 594.462,Z 416.896,A -85,B 0,C 180,E1 -1160.902,E2 -1160.902} C_VEL
LIN {X 0,Y 594.446,Z 425.4,A -85,B 0,C 180,E1 -1161.245,E2 -1161.245} C_VEL
LIN {X 0,Y 594.431,Z 433.729,A -85,B 0,C 180,E1 -1161.673,E2 -1161.673} C_VEL
LIN {X 0,Y 594.368,Z 441.766,A -85,B 0,C 180,E1 -1162.185,E2 -1162.185} C_VEL
LIN {X 0,Y 594.355,Z 449.418,A -85,B 0,C 180,E1 -1162.783,E2 -1162.783} C_VEL
LIN {X 0,Y 594.33,Z 457.809,A -85,B 0,C 180,E1 -1163.589,E2 -1163.589} C_VEL
LIN {X 0,Y 594.309,Z 464.432,A -85,B 0,C 180,E1 -1164.401,E2 -1164.401} C_VEL
LIN {X 0,Y 594.256,Z 469.987,A -85,B 0,C 180,E1 -1165.251,E2 -1165.251} C_VEL
LIN {X 0,Y 594.285,Z 475.147,A -85,B 0,C 180,E1 -1166.271,E2 -1166.271} C_VEL
LIN {X 0,Y 594.245,Z 477.788,A -85,B 0,C 180,E1 -1166.949,E2 -1166.949} C_VEL
LIN {X 0,Y 594.242,Z 480.68,A -85,B 0,C 180,E1 -1167.967,E2 -1167.967} C_VEL
LIN {X 0,Y 594.245,Z 481.935,A -85,B 0,C 180,E1 -1168.645,E2 -1168.645} C_VEL
LIN {X 0,Y 594.235,Z 482.712,A -85,B 0,C 180,E1 -1169.322,E2 -1169.322} C_VEL
LIN {X 0,Y 594.233,Z 483,A -85,B 0,C 180,E1 -1170,E2 -1170} C_VEL
LIN {X 0,Y 594.235,Z 482.712,A -85,B 0,C 180,E1 -1170.678,E2 -1170.678} C_VEL
LIN {X 0,Y 594.245,Z 481.935,A -85,B 0,C 180,E1 -1171.355,E2 -1171.355} C_VEL
LIN {X 0,Y 594.242,Z 480.679,A -85,B 0,C 180,E1 -1172.033,E2 -1172.033} C_VEL
LIN {X 0,Y 594.245,Z 477.787,A -85,B 0,C 180,E1 -1173.051,E2 -1173.051} C_VEL
LIN {X 0,Y 594.285,Z 475.147,A -85,B 0,C 180,E1 -1173.729,E2 -1173.729} C_VEL
LIN {X 0,Y 594.256,Z 469.986,A -85,B 0,C 180,E1 -1174.749,E2 -1174.749} C_VEL
LIN {X 0,Y 594.309,Z 464.431,A -85,B 0,C 180,E1 -1175.599,E2 -1175.599} C_VEL
LIN {X 0,Y 594.344,Z 457.151,A -85,B 0,C 180,E1 -1176.479,E2 -1176.479} C_VEL
LIN {X 0,Y 594.355,Z 449.42,A -85,B 0,C 180,E1 -1177.217,E2 -1177.217} C_VEL
LIN {X 0,Y 594.368,Z 441.768,A -85,B 0,C 180,E1 -1177.815,E2 -1177.815} C_VEL
LIN {X 0,Y 594.431,Z 433.729,A -85,B 0,C 180,E1 -1178.327,E2 -1178.327} C_VEL
LIN {X 0,Y 594.446,Z 425.4,A -85,B 0,C 180,E1 -1178.755,E2 -1178.755} C_VEL
LIN {X 0,Y 594.462,Z 416.898,A -85,B 0,C 180,E1 -1179.098,E2 -1179.098} C_VEL
LIN {X 0,Y 594.497,Z 406.762,A -85,B 0,C 180,E1 -1179.398,E2 -1179.398} C_VEL
LIN {X 0,Y 594.532,Z 395.077,A -85,B 0,C 180,E1 -1179.612,E2 -1179.612} C_VEL
LIN {X 0,Y 594.448,Z 324.754,A -85,B 0,C 180,E1 -1180.462,E2 -1180.462} C_VEL
LIN {X 0,Y 594.335,Z 323.368,A -85,B 0,C 180,E1 -1180.539,E2 -1180.539} C_VEL
LIN {X 0,Y 594.332,Z 309.514,A -85,B 0,C 180,E1 -1182.983,E2 -1182.983} C_VEL
LIN {X 0,Y 594.407,Z 295.85,A -85,B 0,C 180,E1 -1185.428,E2 -1185.428} C_VEL
LIN {X 0,Y 594.473,Z 280.234,A -85,B 0,C 180,E1 -1188.257,E2 -1188.257} C_VEL
LIN {X 0,Y 594.392,Z 271.349,A -85,B 0,C 180,E1 -1189.917,E2 -1189.917} C_VEL
LIN {X 0,Y 594.333,Z 271.255,A -85,B 0,C 180,E1 -1192.968,E2 -1192.968} C_VEL
LIN {X 0,Y 594.357,Z 271.26,A -85,B 0,C 180,E1 -1195.944,E2 -1195.944} C_VEL
LIN {X 0,Y 594.365,Z 271.257,A -85,B 0,C 180,E1 -1198.955,E2 -1198.955} C_VEL
LIN {X 0,Y 594.362,Z 271.262,A -85,B 0,C 180,E1 -1201.64,E2 -1201.64} C_VEL
LIN {X 0,Y 594.352,Z 271.257,A -85,B 0,C 180,E1 -1204.134,E2 -1204.134} C_VEL
LIN {X 0,Y 594.371,Z 271.261,A -85,B 0,C 180,E1 -1207.087,E2 -1207.087} C_VEL
LIN {X 0,Y 594.332,Z 271.262,A -85,B 0,C 180,E1 -1209.769,E2 -1209.769} C_VEL
LIN {X 0,Y 594.327,Z 271.26,A -85,B 0,C 180,E1 -1212.378,E2 -1212.378} C_VEL
LIN {X 0,Y 594.33,Z 271.268,A -85,B 0,C 180,E1 -1215.193,E2 -1215.193} C_VEL
LIN {X 0,Y 594.35,Z 271.257,A -85,B 0,C 180,E1 -1218.154,E2 -1218.154} C_VEL
LIN {X 0,Y 594.345,Z 271.259,A -85,B 0,C 180,E1 -1220.317,E2 -1220.317} C_VEL
LIN {X 0,Y 594.371,Z 271.265,A -85,B 0,C 180,E1 -1222.912,E2 -1222.912} C_VEL
LIN {X 0,Y 594.342,Z 271.258,A -85,B 0,C 180,E1 -1225.865,E2 -1225.865} C_VEL
LIN {X 0,Y 594.351,Z 271.265,A -85,B 0,C 180,E1 -1228.649,E2 -1228.649} C_VEL
LIN {X 0,Y 594.358,Z 271.261,A -85,B 0,C 180,E1 -1231.044,E2 -1231.044} C_VEL
LIN {X 0,Y 594.349,Z 271.258,A -85,B 0,C 180,E1 -1233.299,E2 -1233.299} C_VEL
LIN {X 0,Y 594.321,Z 271.26,A -85,B 0,C 180,E1 -1235.578,E2 -1235.578} C_VEL
LIN {X 0,Y 594.341,Z 271.268,A -85,B 0,C 180,E1 -1238.496,E2 -1238.496} C_VEL
LIN {X 0,Y 594.33,Z 271.259,A -85,B 0,C 180,E1 -1241.381,E2 -1241.381} C_VEL
LIN {X 0,Y 594.328,Z 271.267,A -85,B 0,C 180,E1 -1244.218,E2 -1244.218} C_VEL
LIN {X 0,Y 594.346,Z 271.267,A -85,B 0,C 180,E1 -1246.32,E2 -1246.32} C_VEL
LIN {X 0,Y 594.33,Z 271.26,A -85,B 0,C 180,E1 -1249.094,E2 -1249.094} C_VEL
LIN {X 0,Y 594.36,Z 271.26,A -85,B 0,C 180,E1 -1251.843,E2 -1251.843} C_VEL
LIN {X 0,Y 594.358,Z 271.259,A -85,B 0,C 180,E1 -1254.572,E2 -1254.572} C_VEL
LIN {X 0,Y 594.354,Z 271.257,A -85,B 0,C 180,E1 -1257.289,E2 -1257.289} C_VEL
LIN {X 0,Y 594.401,Z 271.261,A -85,B 0,C 180,E1 -1260,E2 -1260} C_VEL
LIN {X 0,Y 594.352,Z 271.257,A -85,B 0,C 180,E1 -1262.711,E2 -1262.711} C_VEL
LIN {X 0,Y 594.354,Z 271.259,A -85,B 0,C 180,E1 -1265.428,E2 -1265.428} C_VEL
LIN {X 0,Y 594.358,Z 271.261,A -85,B 0,C 180,E1 -1268.158,E2 -1268.158} C_VEL
LIN {X 0,Y 594.332,Z 271.26,A -85,B 0,C 180,E1 -1271.052,E2 -1271.052} C_VEL
LIN {X 0,Y 594.344,Z 271.268,A -85,B 0,C 180,E1 -1273.68,E2 -1273.68} C_VEL
LIN {X 0,Y 594.312,Z 271.264,A -85,B 0,C 180,E1 -1275.285,E2 -1275.285} C_VEL
LIN {X 0,Y 593.64,Z 271.353,A -85,B 0,C 180,E1 -1275.85,E2 -1275.85} C_VEL
LIN {X 0,Y 590.774,Z 271.709,A -85,B 0,C 180,E1 -1276.768,E2 -1276.768} C_VEL
LIN {X 0,Y 588.363,Z 272.012,A -85,B 0,C 180,E1 -1277.506,E2 -1277.506} C_VEL
LIN {X 0,Y 587.339,Z 272.133,A -85,B 0,C 180,E1 -1278.076,E2 -1278.076} C_VEL
LIN {X 0,Y 587.262,Z 272.141,A -85,B 0,C 180,E1 -1278.269,E2 -1278.269} C_VEL
LIN {X 0,Y 587.303,Z 272.138,A -85,B 0,C 180,E1 -1281.039,E2 -1281.039} C_VEL
LIN {X 0,Y 587.271,Z 272.141,A -85,B 0,C 180,E1 -1284.009,E2 -1284.009} C_VEL
LIN {X 0,Y 587.286,Z 272.137,A -85,B 0,C 180,E1 -1286.281,E2 -1286.281} C_VEL
LIN {X 0,Y 587.288,Z 272.144,A -85,B 0,C 180,E1 -1289.125,E2 -1289.125} C_VEL
LIN {X 0,Y 587.304,Z 272.136,A -85,B 0,C 180,E1 -1291.831,E2 -1291.831} C_VEL
LIN {X 0,Y 587.312,Z 272.134,A -85,B 0,C 180,E1 -1294.345,E2 -1294.345} C_VEL
LIN {X 0,Y 587.322,Z 272.135,A -85,B 0,C 180,E1 -1297.609,E2 -1297.609} C_VEL
LIN {X 0,Y 587.283,Z 272.138,A -85,B 0,C 180,E1 -1300.257,E2 -1300.257} C_VEL
LIN {X 0,Y 587.281,Z 272.145,A -85,B 0,C 180,E1 -1303.116,E2 -1303.116} C_VEL
LIN {X 0,Y 587.291,Z 272.136,A -85,B 0,C 180,E1 -1306.048,E2 -1306.048} C_VEL
LIN {X 0,Y 587.302,Z 272.143,A -85,B 0,C 180,E1 -1308.929,E2 -1308.929} C_VEL
LIN {X 0,Y 587.296,Z 272.136,A -85,B 0,C 180,E1 -1311.519,E2 -1311.519} C_VEL
LIN {X 0,Y 587.267,Z 272.141,A -85,B 0,C 180,E1 -1314.099,E2 -1314.099} C_VEL
LIN {X 0,Y 587.326,Z 272.138,A -85,B 0,C 180,E1 -1316.891,E2 -1316.891} C_VEL
LIN {X 0,Y 587.284,Z 272.137,A -85,B 0,C 180,E1 -1319.499,E2 -1319.499} C_VEL
LIN {X 0,Y 587.292,Z 272.143,A -85,B 0,C 180,E1 -1322.318,E2 -1322.318} C_VEL
LIN {X 0,Y 587.319,Z 272.143,A -85,B 0,C 180,E1 -1324.483,E2 -1324.483} C_VEL
LIN {X 0,Y 587.267,Z 272.136,A -85,B 0,C 180,E1 -1327.484,E2 -1327.484} C_VEL
LIN {X 0,Y 587.322,Z 272.276,A -85,B 0,C 180,E1 -1330.061,E2 -1330.061} C_VEL
LIN {X 0,Y 587.522,Z 278.04,A -85,B 0,C 180,E1 -1331.157,E2 -1331.157} C_VEL
LIN {X 0,Y 587.373,Z 293.652,A -85,B 0,C 180,E1 -1334.027,E2 -1334.027} C_VEL
LIN {X 0,Y 587.338,Z 307.313,A -85,B 0,C 180,E1 -1336.507,E2 -1336.507} C_VEL
LIN {X 0,Y 587.269,Z 321.485,A -85,B 0,C 180,E1 -1339.053,E2 -1339.053} C_VEL
LIN {X 0,Y 587.268,Z 323.871,A -85,B 0,C 180,E1 -1339.423,E2 -1339.423} C_VEL
LIN {X 0,Y 587.604,Z 327.205,A -85,B 0,C 180,E1 -1339.493,E2 -1339.493} C_VEL
LIN {X 0,Y 587.535,Z 400.36,A -85,B 0,C 180,E1 -1340.403,E2 -1340.403} C_VEL
LIN {X 0,Y 587.492,Z 410.854,A -85,B 0,C 180,E1 -1340.641,E2 -1340.641} C_VEL
LIN {X 0,Y 587.453,Z 422.564,A -85,B 0,C 180,E1 -1341.053,E2 -1341.053} C_VEL
LIN {X 0,Y 587.395,Z 432.959,A -85,B 0,C 180,E1 -1341.572,E2 -1341.572} C_VEL
LIN {X 0,Y 587.333,Z 441.137,A -85,B 0,C 180,E1 -1342.091,E2 -1342.091} C_VEL
LIN {X 0,Y 587.291,Z 448.893,A -85,B 0,C 180,E1 -1342.695,E2 -1342.695} C_VEL
LIN {X 0,Y 587.286,Z 456.717,A -85,B 0,C 180,E1 -1343.443,E2 -1343.443} C_VEL
LIN {X 0,Y 587.238,Z 464.124,A -85,B 0,C 180,E1 -1344.334,E2 -1344.334} C_VEL
LIN {X 0,Y 587.173,Z 469.736,A -85,B 0,C 180,E1 -1345.194,E2 -1345.194} C_VEL
LIN {X 0,Y 587.211,Z 474.949,A -85,B 0,C 180,E1 -1346.226,E2 -1346.226} C_VEL
LIN {X 0,Y 587.157,Z 477.638,A -85,B 0,C 180,E1 -1346.912,E2 -1346.912} C_VEL
LIN {X 0,Y 587.141,Z 480.575,A -85,B 0,C 180,E1 -1347.942,E2 -1347.942} C_VEL
LIN {X 0,Y 587.144,Z 481.874,A -85,B 0,C 180,E1 -1348.628,E2 -1348.628} C_VEL
LIN {X 0,Y 587.136,Z 482.69,A -85,B 0,C 180,E1 -1349.314,E2 -1349.314} C_VEL
LIN {X 0,Y 587.135,Z 482.996,A -85,B 0,C 180,E1 -1350,E2 -1350} C_VEL
LIN {X 0,Y 587.137,Z 482.733,A -85,B 0,C 180,E1 -1350.686,E2 -1350.686} C_VEL
LIN {X 0,Y 587.146,Z 481.998,A -85,B 0,C 180,E1 -1351.372,E2 -1351.372} C_VEL
LIN {X 0,Y 587.142,Z 480.785,A -85,B 0,C 180,E1 -1352.058,E2 -1352.058} C_VEL
LIN {X 0,Y 587.156,Z 477.938,A -85,B 0,C 180,E1 -1353.088,E2 -1353.088} C_VEL
LIN {X 0,Y 587.211,Z 475.346,A -85,B 0,C 180,E1 -1353.774,E2 -1353.774} C_VEL
LIN {X 0,Y 587.17,Z 470.238,A -85,B 0,C 180,E1 -1354.806,E2 -1354.806} C_VEL
LIN {X 0,Y 587.239,Z 464.741,A -85,B 0,C 180,E1 -1355.666,E2 -1355.666} C_VEL
LIN {X 0,Y 587.268,Z 456.748,A -85,B 0,C 180,E1 -1356.644,E2 -1356.644} C_VEL
LIN {X 0,Y 587.296,Z 448.932,A -85,B 0,C 180,E1 -1357.391,E2 -1357.391} C_VEL
LIN {X 0,Y 587.342,Z 441.184,A -85,B 0,C 180,E1 -1357.996,E2 -1357.996} C_VEL
LIN {X 0,Y 587.395,Z 433.017,A -85,B 0,C 180,E1 -1358.514,E2 -1358.514} C_VEL
LIN {X 0,Y 587.458,Z 422.633,A -85,B 0,C 180,E1 -1359.034,E2 -1359.034} C_VEL
LIN {X 0,Y 587.495,Z 410.973,A -85,B 0,C 180,E1 -1359.445,E2 -1359.445} C_VEL
LIN {X 0,Y 587.543,Z 400.55,A -85,B 0,C 180,E1 -1359.684,E2 -1359.684} C_VEL
LIN {X 0,Y 587.548,Z 348.692,A -85,B 0,C 180,E1 -1360.336,E2 -1360.336} C_VEL
LIN {X 0,Y 587.428,Z 324.91,A -85,B 0,C 180,E1 -1360.631,E2 -1360.631} C_VEL
LIN {X 0,Y 587.256,Z 323.457,A -85,B 0,C 180,E1 -1360.701,E2 -1360.701} C_VEL
LIN {X 0,Y 587.341,Z 307.811,A -85,B 0,C 180,E1 -1363.493,E2 -1363.493} C_VEL
LIN {X 0,Y 587.405,Z 292.192,A -85,B 0,C 180,E1 -1366.329,E2 -1366.329} C_VEL
LIN {X 0,Y 587.501,Z 276.182,A -85,B 0,C 180,E1 -1369.278,E2 -1369.278} C_VEL
LIN {X 0,Y 587.34,Z 272.189,A -85,B 0,C 180,E1 -1370.076,E2 -1370.076} C_VEL
LIN {X 0,Y 587.302,Z 272.129,A -85,B 0,C 180,E1 -1372.864,E2 -1372.864} C_VEL
LIN {X 0,Y 587.324,Z 272.141,A -85,B 0,C 180,E1 -1375.516,E2 -1375.516} C_VEL
LIN {X 0,Y 587.285,Z 272.143,A -85,B 0,C 180,E1 -1377.82,E2 -1377.82} C_VEL
LIN {X 0,Y 587.312,Z 272.134,A -85,B 0,C 180,E1 -1380.505,E2 -1380.505} C_VEL
LIN {X 0,Y 587.319,Z 272.142,A -85,B 0,C 180,E1 -1383.397,E2 -1383.397} C_VEL
LIN {X 0,Y 587.27,Z 272.141,A -85,B 0,C 180,E1 -1385.901,E2 -1385.901} C_VEL
LIN {X 0,Y 587.305,Z 272.135,A -85,B 0,C 180,E1 -1388.48,E2 -1388.48} C_VEL
LIN {X 0,Y 587.323,Z 272.141,A -85,B 0,C 180,E1 -1391.157,E2 -1391.157} C_VEL
LIN {X 0,Y 587.296,Z 272.136,A -85,B 0,C 180,E1 -1394.11,E2 -1394.11} C_VEL
LIN {X 0,Y 587.283,Z 272.146,A -85,B 0,C 180,E1 -1396.991,E2 -1396.991} C_VEL
LIN {X 0,Y 587.294,Z 272.137,A -85,B 0,C 180,E1 -1399.744,E2 -1399.744} C_VEL
LIN {X 0,Y 587.328,Z 272.133,A -85,B 0,C 180,E1 -1402.391,E2 -1402.391} C_VEL
LIN {X 0,Y 587.315,Z 272.134,A -85,B 0,C 180,E1 -1405.655,E2 -1405.655} C_VEL
LIN {X 0,Y 587.322,Z 272.134,A -85,B 0,C 180,E1 -1408.23,E2 -1408.23} C_VEL
LIN {X 0,Y 587.327,Z 272.14,A -85,B 0,C 180,E1 -1410.868,E2 -1410.868} C_VEL
LIN {X 0,Y 587.302,Z 272.135,A -85,B 0,C 180,E1 -1413.828,E2 -1413.828} C_VEL
LIN {X 0,Y 587.282,Z 272.145,A -85,B 0,C 180,E1 -1416.74,E2 -1416.74} C_VEL
LIN {X 0,Y 587.301,Z 272.139,A -85,B 0,C 180,E1 -1418.967,E2 -1418.967} C_VEL
LIN {X 0,Y 587.308,Z 272.135,A -85,B 0,C 180,E1 -1421.15,E2 -1421.15} C_VEL
LIN {X 0,Y 587.277,Z 272.142,A -85,B 0,C 180,E1 -1424.023,E2 -1424.023} C_VEL
LIN {X 0,Y 587.321,Z 272.139,A -85,B 0,C 180,E1 -1426.153,E2 -1426.153} C_VEL
LIN {X 0,Y 587.325,Z 272.133,A -85,B 0,C 180,E1 -1428.962,E2 -1428.962} C_VEL
LIN {X 0,Y 587.319,Z 272.135,A -85,B 0,C 180,E1 -1431.744,E2 -1431.744} C_VEL
LIN {X 0,Y 587.328,Z 272.136,A -85,B 0,C 180,E1 -1434.507,E2 -1434.507} C_VEL
LIN {X 0,Y 587.322,Z 272.133,A -85,B 0,C 180,E1 -1437.256,E2 -1437.256} C_VEL
LIN {X 0,Y 587.369,Z 272.137,A -85,B 0,C 180,E1 -1440,E2 -1440} C_VEL
LIN {X 0,Y 587.32,Z 272.133,A -85,B 0,C 180,E1 -1442.743,E2 -1442.743} C_VEL
LIN {X 0,Y 587.324,Z 272.136,A -85,B 0,C 180,E1 -1445.493,E2 -1445.493} C_VEL
LIN {X 0,Y 587.314,Z 272.137,A -85,B 0,C 180,E1 -1448.256,E2 -1448.256} C_VEL
LIN {X 0,Y 587.302,Z 272.136,A -85,B 0,C 180,E1 -1451.117,E2 -1451.117} C_VEL
LIN {X 0,Y 587.32,Z 272.14,A -85,B 0,C 180,E1 -1453.847,E2 -1453.847} C_VEL
LIN {X 0,Y 587.279,Z 272.138,A -85,B 0,C 180,E1 -1456.796,E2 -1456.796} C_VEL
LIN {X 0,Y 587.285,Z 272.147,A -85,B 0,C 180,E1 -1459.577,E2 -1459.577} C_VEL
LIN {X 0,Y 587.287,Z 272.142,A -85,B 0,C 180,E1 -1461.776,E2 -1461.776} C_VEL
LIN {X 0,Y 587.288,Z 272.138,A -85,B 0,C 180,E1 -1464.761,E2 -1464.761} C_VEL
LIN {X 0,Y 587.284,Z 272.142,A -85,B 0,C 180,E1 -1467.683,E2 -1467.683} C_VEL
LIN {X 0,Y 587.282,Z 272.137,A -85,B 0,C 180,E1 -1470.173,E2 -1470.173} C_VEL
LIN {X 0,Y 587.312,Z 272.135,A -85,B 0,C 180,E1 -1472.581,E2 -1472.581} C_VEL
LIN {X 0,Y 587.29,Z 272.145,A -85,B 0,C 180,E1 -1475.058,E2 -1475.058} C_VEL
LIN {X 0,Y 587.314,Z 272.134,A -85,B 0,C 180,E1 -1477.837,E2 -1477.837} C_VEL
LIN {X 0,Y 587.284,Z 272.138,A -85,B 0,C 180,E1 -1480.257,E2 -1480.257} C_VEL
LIN {X 0,Y 587.282,Z 272.145,A -85,B 0,C 180,E1 -1483.116,E2 -1483.116} C_VEL
LIN {X 0,Y 587.291,Z 272.137,A -85,B 0,C 180,E1 -1486.048,E2 -1486.048} C_VEL
LIN {X 0,Y 587.302,Z 272.143,A -85,B 0,C 180,E1 -1488.929,E2 -1488.929} C_VEL
LIN {X 0,Y 587.296,Z 272.136,A -85,B 0,C 180,E1 -1491.519,E2 -1491.519} C_VEL
LIN {X 0,Y 587.268,Z 272.141,A -85,B 0,C 180,E1 -1494.099,E2 -1494.099} C_VEL
LIN {X 0,Y 587.326,Z 272.137,A -85,B 0,C 180,E1 -1496.89,E2 -1496.89} C_VEL
LIN {X 0,Y 587.3,Z 272.135,A -85,B 0,C 180,E1 -1499.496,E2 -1499.496} C_VEL
LIN {X 0,Y 587.282,Z 272.137,A -85,B 0,C 180,E1 -1501.402,E2 -1501.402} C_VEL
LIN {X 0,Y 587.3,Z 272.137,A -85,B 0,C 180,E1 -1503.831,E2 -1503.831} C_VEL
LIN {X 0,Y 587.291,Z 272.137,A -85,B 0,C 180,E1 -1506.741,E2 -1506.741} C_VEL
LIN {X 0,Y 587.31,Z 272.138,A -85,B 0,C 180,E1 -1509.695,E2 -1509.695} C_VEL
LIN {X 0,Y 587.399,Z 272.466,A -85,B 0,C 180,E1 -1510.063,E2 -1510.063} C_VEL
LIN {X 0,Y 587.465,Z 282.186,A -85,B 0,C 180,E1 -1511.878,E2 -1511.878} C_VEL
LIN {X 0,Y 587.379,Z 297.802,A -85,B 0,C 180,E1 -1514.739,E2 -1514.739} C_VEL
LIN {X 0,Y 587.308,Z 313.418,A -85,B 0,C 180,E1 -1517.562,E2 -1517.562} C_VEL
LIN {X 0,Y 587.25,Z 323.609,A -85,B 0,C 180,E1 -1519.358,E2 -1519.358} C_VEL
LIN {X 0,Y 587.497,Z 325.588,A -85,B 0,C 180,E1 -1519.427,E2 -1519.427} C_VEL
LIN {X 0,Y 587.541,Z 399.153,A -85,B 0,C 180,E1 -1520.338,E2 -1520.338} C_VEL
LIN {X 0,Y 587.5,Z 408.422,A -85,B 0,C 180,E1 -1520.533,E2 -1520.533} C_VEL
LIN {X 0,Y 587.446,Z 416.898,A -85,B 0,C 180,E1 -1520.793,E2 -1520.793} C_VEL
LIN {X 0,Y 587.418,Z 425.403,A -85,B 0,C 180,E1 -1521.139,E2 -1521.139} C_VEL
LIN {X 0,Y 587.394,Z 433.732,A -85,B 0,C 180,E1 -1521.572,E2 -1521.572} C_VEL
LIN {X 0,Y 587.335,Z 441.768,A -85,B 0,C 180,E1 -1522.091,E2 -1522.091} C_VEL
LIN {X 0,Y 587.29,Z 449.418,A -85,B 0,C 180,E1 -1522.695,E2 -1522.695} C_VEL
LIN {X 0,Y 587.281,Z 457.809,A -85,B 0,C 180,E1 -1523.512,E2 -1523.512} C_VEL
LIN {X 0,Y 587.238,Z 464.433,A -85,B 0,C 180,E1 -1524.334,E2 -1524.334} C_VEL
LIN {X 0,Y 587.17,Z 469.987,A -85,B 0,C 180,E1 -1525.194,E2 -1525.194} C_VEL
LIN {X 0,Y 587.21,Z 475.148,A -85,B 0,C 180,E1 -1526.226,E2 -1526.226} C_VEL
LIN {X 0,Y 587.155,Z 477.788,A -85,B 0,C 180,E1 -1526.912,E2 -1526.912} C_VEL
LIN {X 0,Y 587.141,Z 480.68,A -85,B 0,C 180,E1 -1527.942,E2 -1527.942} C_VEL
LIN {X 0,Y 587.145,Z 481.936,A -85,B 0,C 180,E1 -1528.628,E2 -1528.628} C_VEL
LIN {X 0,Y 587.136,Z 482.712,A -85,B 0,C 180,E1 -1529.314,E2 -1529.314} C_VEL
LIN {X 0,Y 587.134,Z 483,A -85,B 0,C 180,E1 -1530,E2 -1530} C_VEL
LIN {X 0,Y 587.136,Z 482.711,A -85,B 0,C 180,E1 -1530.686,E2 -1530.686} C_VEL
LIN {X 0,Y 587.145,Z 481.936,A -85,B 0,C 180,E1 -1531.372,E2 -1531.372} C_VEL
LIN {X 0,Y 587.141,Z 480.68,A -85,B 0,C 180,E1 -1532.058,E2 -1532.058} C_VEL
LIN {X 0,Y 587.155,Z 477.788,A -85,B 0,C 180,E1 -1533.088,E2 -1533.088} C_VEL
LIN {X 0,Y 587.21,Z 475.148,A -85,B 0,C 180,E1 -1533.774,E2 -1533.774} C_VEL
LIN {X 0,Y 587.17,Z 469.986,A -85,B 0,C 180,E1 -1534.806,E2 -1534.806} C_VEL
LIN {X 0,Y 587.253,Z 463.189,A -85,B 0,C 180,E1 -1535.838,E2 -1535.838} C_VEL
LIN {X 0,Y 587.269,Z 456.287,A -85,B 0,C 180,E1 -1536.645,E2 -1536.645} C_VEL
LIN {X 0,Y 587.294,Z 448.407,A -85,B 0,C 180,E1 -1537.391,E2 -1537.391} C_VEL
LIN {X 0,Y 587.341,Z 440.552,A -85,B 0,C 180,E1 -1537.996,E2 -1537.996} C_VEL
LIN {X 0,Y 587.435,Z 430.738,A -85,B 0,C 180,E1 -1538.601,E2 -1538.601} C_VEL
LIN {X 0,Y 587.464,Z 419.306,A -85,B 0,C 180,E1 -1539.12,E2 -1539.12} C_VEL
LIN {X 0,Y 587.512,Z 409.254,A -85,B 0,C 180,E1 -1539.445,E2 -1539.445} C_VEL
LIN {X 0,Y 587.538,Z 400.458,A -85,B 0,C 180,E1 -1539.64,E2 -1539.64} C_VEL
LIN {X 0,Y 587.603,Z 336.173,A -85,B 0,C 180,E1 -1540.442,E2 -1540.442} C_VEL
LIN {X 0,Y 587.325,Z 324.375,A -85,B 0,C 180,E1 -1540.598,E2 -1540.598} C_VEL
LIN {X 0,Y 587.248,Z 323.259,A -85,B 0,C 180,E1 -1540.685,E2 -1540.685} C_VEL
LIN {X 0,Y 587.283,Z 309.514,A -85,B 0,C 180,E1 -1543.142,E2 -1543.142} C_VEL
LIN {X 0,Y 587.389,Z 295.85,A -85,B 0,C 180,E1 -1545.617,E2 -1545.617} C_VEL
LIN {X 0,Y 587.487,Z 280.234,A -85,B 0,C 180,E1 -1548.482,E2 -1548.482} C_VEL
LIN {X 0,Y 587.344,Z 272.274,A -85,B 0,C 180,E1 -1549.984,E2 -1549.984} C_VEL
LIN {X 0,Y 587.284,Z 272.131,A -85,B 0,C 180,E1 -1552.86,E2 -1552.86} C_VEL
LIN {X 0,Y 587.321,Z 272.142,A -85,B 0,C 180,E1 -1555.517,E2 -1555.517} C_VEL
LIN {X 0,Y 587.283,Z 272.143,A -85,B 0,C 180,E1 -1557.82,E2 -1557.82} C_VEL
LIN {X 0,Y 587.29,Z 272.137,A -85,B 0,C 180,E1 -1560.172,E2 -1560.172} C_VEL
LIN {X 0,Y 587.318,Z 272.133,A -85,B 0,C 180,E1 -1562.579,E2 -1562.579} C_VEL
LIN {X 0,Y 587.294,Z 272.141,A -85,B 0,C 180,E1 -1565.057,E2 -1565.057} C_VEL
LIN {X 0,Y 587.309,Z 272.136,A -85,B 0,C 180,E1 -1567.835,E2 -1567.835} C_VEL
LIN {X 0,Y 587.286,Z 272.137,A -85,B 0,C 180,E1 -1570.256,E2 -1570.256} C_VEL
LIN {X 0,Y 587.283,Z 272.147,A -85,B 0,C 180,E1 -1573.115,E2 -1573.115} C_VEL
LIN {X 0,Y 587.289,Z 272.136,A -85,B 0,C 180,E1 -1576.046,E2 -1576.046} C_VEL
LIN {X 0,Y 587.324,Z 272.141,A -85,B 0,C 180,E1 -1578.925,E2 -1578.925} C_VEL
LIN {X 0,Y 587.302,Z 272.137,A -85,B 0,C 180,E1 -1581.519,E2 -1581.519} C_VEL
LIN {X 0,Y 587.264,Z 272.14,A -85,B 0,C 180,E1 -1584.098,E2 -1584.098} C_VEL
LIN {X 0,Y 587.32,Z 272.142,A -85,B 0,C 180,E1 -1586.889,E2 -1586.889} C_VEL
LIN {X 0,Y 587.295,Z 272.136,A -85,B 0,C 180,E1 -1589.495,E2 -1589.495} C_VEL
LIN {X 0,Y 587.276,Z 272.139,A -85,B 0,C 180,E1 -1591.401,E2 -1591.401} C_VEL
LIN {X 0,Y 587.301,Z 272.135,A -85,B 0,C 180,E1 -1593.828,E2 -1593.828} C_VEL
LIN {X 0,Y 587.282,Z 272.145,A -85,B 0,C 180,E1 -1596.74,E2 -1596.74} C_VEL
LIN {X 0,Y 587.301,Z 272.138,A -85,B 0,C 180,E1 -1598.967,E2 -1598.967} C_VEL
LIN {X 0,Y 587.308,Z 272.135,A -85,B 0,C 180,E1 -1601.15,E2 -1601.15} C_VEL
LIN {X 0,Y 587.276,Z 272.142,A -85,B 0,C 180,E1 -1604.024,E2 -1604.024} C_VEL
LIN {X 0,Y 587.321,Z 272.139,A -85,B 0,C 180,E1 -1606.153,E2 -1606.153} C_VEL
LIN {X 0,Y 587.324,Z 272.133,A -85,B 0,C 180,E1 -1608.962,E2 -1608.962} C_VEL
LIN {X 0,Y 587.319,Z 272.136,A -85,B 0,C 180,E1 -1611.744,E2 -1611.744} C_VEL
LIN {X 0,Y 587.328,Z 272.136,A -85,B 0,C 180,E1 -1614.507,E2 -1614.507} C_VEL
LIN {X 0,Y 587.322,Z 272.133,A -85,B 0,C 180,E1 -1617.257,E2 -1617.257} C_VEL
LIN {X 0,Y 587.369,Z 272.137,A -85,B 0,C 180,E1 -1620,E2 -1620} C_VEL
LIN {X 0,Y 587.32,Z 272.133,A -85,B 0,C 180,E1 -1622.744,E2 -1622.744} C_VEL
LIN {X 0,Y 587.325,Z 272.136,A -85,B 0,C 180,E1 -1625.493,E2 -1625.493} C_VEL
LIN {X 0,Y 587.314,Z 272.137,A -85,B 0,C 180,E1 -1628.256,E2 -1628.256} C_VEL
LIN {X 0,Y 587.302,Z 272.136,A -85,B 0,C 180,E1 -1631.117,E2 -1631.117} C_VEL
LIN {X 0,Y 587.319,Z 272.14,A -85,B 0,C 180,E1 -1633.847,E2 -1633.847} C_VEL
LIN {X 0,Y 587.279,Z 272.138,A -85,B 0,C 180,E1 -1636.796,E2 -1636.796} C_VEL
LIN {X 0,Y 587.262,Z 272.141,A -85,B 0,C 180,E1 -1638.269,E2 -1638.269} C_VEL
LIN {X 0,Y 586.612,Z 272.222,A -85,B 0,C 180,E1 -1638.841,E2 -1638.841} C_VEL
LIN {X 0,Y 583.766,Z 272.582,A -85,B 0,C 180,E1 -1639.77,E2 -1639.77} C_VEL
LIN {X 0,Y 581.36,Z 272.878,A -85,B 0,C 180,E1 -1640.517,E2 -1640.517} C_VEL
LIN {X 0,Y 580.338,Z 273.006,A -85,B 0,C 180,E1 -1641.093,E2 -1641.093} C_VEL
LIN {X 0,Y 580.261,Z 273.018,A -85,B 0,C 180,E1 -1641.289,E2 -1641.289} C_VEL
LIN {X 0,Y 580.235,Z 273.015,A -85,B 0,C 180,E1 -1644.319,E2 -1644.319} C_VEL
LIN {X 0,Y 580.233,Z 273.016,A -85,B 0,C 180,E1 -1646.626,E2 -1646.626} C_VEL
LIN {X 0,Y 580.237,Z 273.025,A -85,B 0,C 180,E1 -1649.301,E2 -1649.301} C_VEL
LIN {X 0,Y 580.272,Z 273.011,A -85,B 0,C 180,E1 -1652.202,E2 -1652.202} C_VEL
LIN {X 0,Y 580.262,Z 273.015,A -85,B 0,C 180,E1 -1654.698,E2 -1654.698} C_VEL
LIN {X 0,Y 580.273,Z 273.018,A -85,B 0,C 180,E1 -1657.27,E2 -1657.27} C_VEL
LIN {X 0,Y 580.264,Z 273.012,A -85,B 0,C 180,E1 -1660.269,E2 -1660.269} C_VEL
LIN {X 0,Y 580.226,Z 273.02,A -85,B 0,C 180,E1 -1663.387,E2 -1663.387} C_VEL
LIN {X 0,Y 580.243,Z 273.015,A -85,B 0,C 180,E1 -1665.612,E2 -1665.612} C_VEL
LIN {X 0,Y 580.233,Z 273.017,A -85,B 0,C 180,E1 -1668.228,E2 -1668.228} C_VEL
LIN {X 0,Y 580.255,Z 273.02,A -85,B 0,C 180,E1 -1670.964,E2 -1670.964} C_VEL
LIN {X 0,Y 580.236,Z 273.015,A -85,B 0,C 180,E1 -1673.595,E2 -1673.595} C_VEL
LIN {X 0,Y 580.263,Z 273.014,A -85,B 0,C 180,E1 -1676.143,E2 -1676.143} C_VEL
LIN {X 0,Y 580.256,Z 273.023,A -85,B 0,C 180,E1 -1678.614,E2 -1678.614} C_VEL
LIN {X 0,Y 580.242,Z 273.017,A -85,B 0,C 180,E1 -1681.022,E2 -1681.022} C_VEL
LIN {X 0,Y 580.264,Z 273.012,A -85,B 0,C 180,E1 -1683.672,E2 -1683.672} C_VEL
LIN {X 0,Y 580.24,Z 273.02,A -85,B 0,C 180,E1 -1686.441,E2 -1686.441} C_VEL
LIN {X 0,Y 580.248,Z 273.017,A -85,B 0,C 180,E1 -1689.437,E2 -1689.437} C_VEL
LIN {X 0,Y 580.31,Z 273.224,A -85,B 0,C 180,E1 -1689.994,E2 -1689.994} C_VEL
LIN {X 0,Y 580.504,Z 279.994,A -85,B 0,C 180,E1 -1691.287,E2 -1691.287} C_VEL
LIN {X 0,Y 580.358,Z 295.606,A -85,B 0,C 180,E1 -1694.189,E2 -1694.189} C_VEL
LIN {X 0,Y 580.236,Z 311.219,A -85,B 0,C 180,E1 -1697.052,E2 -1697.052} C_VEL
LIN {X 0,Y 580.2,Z 323.733,A -85,B 0,C 180,E1 -1699.282,E2 -1699.282} C_VEL
LIN {X 0,Y 580.647,Z 327.352,A -85,B 0,C 180,E1 -1699.367,E2 -1699.367} C_VEL
LIN {X 0,Y 580.554,Z 400.392,A -85,B 0,C 180,E1 -1700.287,E2 -1700.287} C_VEL
LIN {X 0,Y 580.499,Z 410.875,A -85,B 0,C 180,E1 -1700.528,E2 -1700.528} C_VEL
LIN {X 0,Y 580.435,Z 422.574,A -85,B 0,C 180,E1 -1700.944,E2 -1700.944} C_VEL
LIN {X 0,Y 580.362,Z 432.966,A -85,B 0,C 180,E1 -1701.469,E2 -1701.469} C_VEL
LIN {X 0,Y 580.285,Z 441.147,A -85,B 0,C 180,E1 -1701.994,E2 -1701.994} C_VEL
LIN {X 0,Y 580.24,Z 448.901,A -85,B 0,C 180,E1 -1702.606,E2 -1702.606} C_VEL
LIN {X 0,Y 580.21,Z 456.515,A -85,B 0,C 180,E1 -1703.342,E2 -1703.342} C_VEL
LIN {X 0,Y 580.173,Z 464.128,A -85,B 0,C 180,E1 -1704.265,E2 -1704.265} C_VEL
LIN {X 0,Y 580.088,Z 469.739,A -85,B 0,C 180,E1 -1705.135,E2 -1705.135} C_VEL
LIN {X 0,Y 580.138,Z 474.952,A -85,B 0,C 180,E1 -1706.18,E2 -1706.18} C_VEL
LIN {X 0,Y 580.072,Z 477.639,A -85,B 0,C 180,E1 -1706.875,E2 -1706.875} C_VEL
LIN {X 0,Y 580.041,Z 480.577,A -85,B 0,C 180,E1 -1707.917,E2 -1707.917} C_VEL
LIN {X 0,Y 580.044,Z 481.873,A -85,B 0,C 180,E1 -1708.611,E2 -1708.611} C_VEL
LIN {X 0,Y 580.036,Z 482.69,A -85,B 0,C 180,E1 -1709.306,E2 -1709.306} C_VEL
LIN {X 0,Y 580.036,Z 482.996,A -85,B 0,C 180,E1 -1710,E2 -1710} C_VEL
LIN {X 0,Y 580.037,Z 482.731,A -85,B 0,C 180,E1 -1710.694,E2 -1710.694} C_VEL
LIN {X 0,Y 580.046,Z 481.998,A -85,B 0,C 180,E1 -1711.389,E2 -1711.389} C_VEL
LIN {X 0,Y 580.041,Z 480.785,A -85,B 0,C 180,E1 -1712.083,E2 -1712.083} C_VEL
LIN {X 0,Y 580.071,Z 477.937,A -85,B 0,C 180,E1 -1713.125,E2 -1713.125} C_VEL
LIN {X 0,Y 580.123,Z 475.344,A -85,B 0,C 180,E1 -1713.82,E2 -1713.82} C_VEL
LIN {X 0,Y 580.075,Z 470.235,A -85,B 0,C 180,E1 -1714.865,E2 -1714.865} C_VEL
LIN {X 0,Y 580.174,Z 464.738,A -85,B 0,C 180,E1 -1715.735,E2 -1715.735} C_VEL
LIN {X 0,Y 580.195,Z 457.506,A -85,B 0,C 180,E1 -1716.645,E2 -1716.645} C_VEL
LIN {X 0,Y 580.254,Z 448.927,A -85,B 0,C 180,E1 -1717.481,E2 -1717.481} C_VEL
LIN {X 0,Y 580.308,Z 441.178,A -85,B 0,C 180,E1 -1718.093,E2 -1718.093} C_VEL
LIN {X 0,Y 580.36,Z 433.005,A -85,B 0,C 180,E1 -1718.618,E2 -1718.618} C_VEL
LIN {X 0,Y 580.437,Z 422.619,A -85,B 0,C 180,E1 -1719.144,E2 -1719.144} C_VEL
LIN {X 0,Y 580.513,Z 410.952,A -85,B 0,C 180,E1 -1719.56,E2 -1719.56} C_VEL
LIN {X 0,Y 580.563,Z 400.516,A -85,B 0,C 180,E1 -1719.801,E2 -1719.801} C_VEL
LIN {X 0,Y 580.6,Z 342.427,A -85,B 0,C 180,E1 -1720.538,E2 -1720.538} C_VEL
LIN {X 0,Y 580.402,Z 325.515,A -85,B 0,C 180,E1 -1720.75,E2 -1720.75} C_VEL
LIN {X 0,Y 580.232,Z 323.813,A -85,B 0,C 180,E1 -1720.803,E2 -1720.803} C_VEL
LIN {X 0,Y 580.226,Z 319.522,A -85,B 0,C 180,E1 -1721.528,E2 -1721.528} C_VEL
LIN {X 0,Y 580.294,Z 303.521,A -85,B 0,C 180,E1 -1724.445,E2 -1724.445} C_VEL
LIN {X 0,Y 580.404,Z 287.405,A -85,B 0,C 180,E1 -1727.421,E2 -1727.421} C_VEL
LIN {X 0,Y 580.464,Z 274.617,A -85,B 0,C 180,E1 -1729.816,E2 -1729.816} C_VEL
LIN {X 0,Y 580.33,Z 273.082,A -85,B 0,C 180,E1 -1730.144,E2 -1730.144} C_VEL
LIN {X 0,Y 580.253,Z 273.007,A -85,B 0,C 180,E1 -1732.999,E2 -1732.999} C_VEL
LIN {X 0,Y 580.26,Z 273.018,A -85,B 0,C 180,E1 -1735.85,E2 -1735.85} C_VEL
LIN {X 0,Y 580.273,Z 273.012,A -85,B 0,C 180,E1 -1738.976,E2 -1738.976} C_VEL
LIN {X 0,Y 580.263,Z 273.02,A -85,B 0,C 180,E1 -1741.385,E2 -1741.385} C_VEL
LIN {X 0,Y 580.269,Z 273.014,A -85,B 0,C 180,E1 -1743.857,E2 -1743.857} C_VEL
LIN {X 0,Y 580.271,Z 273.014,A -85,B 0,C 180,E1 -1746.93,E2 -1746.93} C_VEL
LIN {X 0,Y 580.264,Z 273.013,A -85,B 0,C 180,E1 -1749.934,E2 -1749.934} C_VEL
LIN {X 0,Y 580.246,Z 273.016,A -85,B 0,C 180,E1 -1752.708,E2 -1752.708} C_VEL
LIN {X 0,Y 580.243,Z 273.017,A -85,B 0,C 180,E1 -1755.61,E2 -1755.61} C_VEL
LIN {X 0,Y 580.262,Z 273.016,A -85,B 0,C 180,E1 -1758.669,E2 -1758.669} C_VEL
LIN {X 0,Y 580.258,Z 273.022,A -85,B 0,C 180,E1 -1760.963,E2 -1760.963} C_VEL
LIN {X 0,Y 580.235,Z 273.016,A -85,B 0,C 180,E1 -1763.594,E2 -1763.594} C_VEL
LIN {X 0,Y 580.26,Z 273.013,A -85,B 0,C 180,E1 -1766.141,E2 -1766.141} C_VEL
LIN {X 0,Y 580.255,Z 273.02,A -85,B 0,C 180,E1 -1768.613,E2 -1768.613} C_VEL
LIN {X 0,Y 580.265,Z 273.017,A -85,B 0,C 180,E1 -1771.022,E2 -1771.022} C_VEL
LIN {X 0,Y 580.257,Z 273.012,A -85,B 0,C 180,E1 -1773.67,E2 -1773.67} C_VEL
LIN {X 0,Y 580.235,Z 273.022,A -85,B 0,C 180,E1 -1776.44,E2 -1776.44} C_VEL
LIN {X 0,Y 580.239,Z 273.015,A -85,B 0,C 180,E1 -1779.436,E2 -1779.436} C_VEL
LIN {X 0,Y 580.223,Z 273.017,A -85,B 0,C 180,E1 -1781.643,E2 -1781.643} C_VEL
LIN {X 0,Y 580.255,Z 273.021,A -85,B 0,C 180,E1 -1784.546,E2 -1784.546} C_VEL
LIN {X 0,Y 580.222,Z 273.021,A -85,B 0,C 180,E1 -1786.695,E2 -1786.695} C_VEL
LIN {X 0,Y 580.293,Z 273.01,A -85,B 0,C 180,E1 -1788.827,E2 -1788.827} C_VEL
LIN {X 0,Y 580.287,Z 273.01,A -85,B 0,C 180,E1 -1791.643,E2 -1791.643} C_VEL
LIN {X 0,Y 580.297,Z 273.013,A -85,B 0,C 180,E1 -1794.44,E2 -1794.44} C_VEL
LIN {X 0,Y 580.332,Z 273.011,A -85,B 0,C 180,E1 -1797.918,E2 -1797.918} C_VEL
LIN {X 0,Y 580.337,Z 273.012,A -85,B 0,C 180,E1 -1800,E2 -1800} C_VEL
LIN {X 0,Y 580.289,Z 273.009,A -85,B 0,C 180,E1 -1802.777,E2 -1802.777} C_VEL
LIN {X 0,Y 580.294,Z 273.013,A -85,B 0,C 180,E1 -1805.56,E2 -1805.56} C_VEL
LIN {X 0,Y 580.28,Z 273.012,A -85,B 0,C 180,E1 -1808.357,E2 -1808.357} C_VEL
LIN {X 0,Y 580.254,Z 273.015,A -85,B 0,C 180,E1 -1811.174,E2 -1811.174} C_VEL
LIN {X 0,Y 580.279,Z 273.014,A -85,B 0,C 180,E1 -1814.018,E2 -1814.018} C_VEL
LIN {X 0,Y 580.237,Z 273.016,A -85,B 0,C 180,E1 -1816.899,E2 -1816.899} C_VEL
LIN {X 0,Y 580.258,Z 273.017,A -85,B 0,C 180,E1 -1819.824,E2 -1819.824} C_VEL
LIN {X 0,Y 580.221,Z 273.019,A -85,B 0,C 180,E1 -1822.055,E2 -1822.055} C_VEL
LIN {X 0,Y 580.267,Z 273.016,A -85,B 0,C 180,E1 -1825.082,E2 -1825.082} C_VEL
LIN {X 0,Y 580.229,Z 273.018,A -85,B 0,C 180,E1 -1827.848,E2 -1827.848} C_VEL
LIN {X 0,Y 580.247,Z 273.016,A -85,B 0,C 180,E1 -1830.691,E2 -1830.691} C_VEL
LIN {X 0,Y 580.266,Z 273.019,A -85,B 0,C 180,E1 -1833.313,E2 -1833.313} C_VEL
LIN {X 0,Y 580.214,Z 273.019,A -85,B 0,C 180,E1 -1835.754,E2 -1835.754} C_VEL
LIN {X 0,Y 580.269,Z 273.011,A -85,B 0,C 180,E1 -1838.148,E2 -1838.148} C_VEL
LIN {X 0,Y 580.28,Z 273.017,A -85,B 0,C 180,E1 -1840.845,E2 -1840.845} C_VEL
LIN {X 0,Y 580.228,Z 273.017,A -85,B 0,C 180,E1 -1843.663,E2 -1843.663} C_VEL
LIN {X 0,Y 580.227,Z 273.022,A -85,B 0,C 180,E1 -1846.615,E2 -1846.615} C_VEL
LIN {X 0,Y 580.249,Z 273.018,A -85,B 0,C 180,E1 -1849.154,E2 -1849.154} C_VEL
LIN {X 0,Y 580.27,Z 273.011,A -85,B 0,C 180,E1 -1851.93,E2 -1851.93} C_VEL
LIN {X 0,Y 580.219,Z 273.024,A -85,B 0,C 180,E1 -1854.451,E2 -1854.451} C_VEL
LIN {X 0,Y 580.277,Z 273.014,A -85,B 0,C 180,E1 -1856.975,E2 -1856.975} C_VEL
LIN {X 0,Y 580.263,Z 273.012,A -85,B 0,C 180,E1 -1859.424,E2 -1859.424} C_VEL
LIN {X 0,Y 580.236,Z 273.02,A -85,B 0,C 180,E1 -1862.153,E2 -1862.153} C_VEL
LIN {X 0,Y 580.277,Z 273.013,A -85,B 0,C 180,E1 -1864.92,E2 -1864.92} C_VEL
LIN {X 0,Y 580.237,Z 273.015,A -85,B 0,C 180,E1 -1867.947,E2 -1867.947} C_VEL
LIN {X 0,Y 580.304,Z 273.22,A -85,B 0,C 180,E1 -1869.947,E2 -1869.947} C_VEL
LIN {X 0,Y 580.503,Z 280.234,A -85,B 0,C 180,E1 -1871.287,E2 -1871.287} C_VEL
LIN {X 0,Y 580.355,Z 295.85,A -85,B 0,C 180,E1 -1874.189,E2 -1874.189} C_VEL
LIN {X 0,Y 580.235,Z 311.466,A -85,B 0,C 180,E1 -1877.052,E2 -1877.052} C_VEL
LIN {X 0,Y 580.191,Z 323.588,A -85,B 0,C 180,E1 -1879.225,E2 -1879.225} C_VEL
LIN {X 0,Y 580.43,Z 325.562,A -85,B 0,C 180,E1 -1879.296,E2 -1879.296} C_VEL
LIN {X 0,Y 580.58,Z 362.881,A -85,B 0,C 180,E1 -1879.759,E2 -1879.759} C_VEL
LIN {X 0,Y 580.558,Z 400.451,A -85,B 0,C 180,E1 -1880.243,E2 -1880.243} C_VEL
LIN {X 0,Y 580.51,Z 410.913,A -85,B 0,C 180,E1 -1880.484,E2 -1880.484} C_VEL
LIN {X 0,Y 580.46,Z 421.617,A -85,B 0,C 180,E1 -1880.856,E2 -1880.856} C_VEL
LIN {X 0,Y 580.365,Z 432.235,A -85,B 0,C 180,E1 -1881.382,E2 -1881.382} C_VEL
LIN {X 0,Y 580.307,Z 440.546,A -85,B 0,C 180,E1 -1881.907,E2 -1881.907} C_VEL
LIN {X 0,Y 580.252,Z 448.405,A -85,B 0,C 180,E1 -1882.519,E2 -1882.519} C_VEL
LIN {X 0,Y 580.227,Z 455.465,A -85,B 0,C 180,E1 -1883.189,E2 -1883.189} C_VEL
LIN {X 0,Y 580.193,Z 463.191,A -85,B 0,C 180,E1 -1884.09,E2 -1884.09} C_VEL
LIN {X 0,Y 580.084,Z 469.988,A -85,B 0,C 180,E1 -1885.135,E2 -1885.135} C_VEL
LIN {X 0,Y 580.137,Z 475.148,A -85,B 0,C 180,E1 -1886.18,E2 -1886.18} C_VEL
LIN {X 0,Y 580.07,Z 477.789,A -85,B 0,C 180,E1 -1886.875,E2 -1886.875} C_VEL
LIN {X 0,Y 580.041,Z 480.681,A -85,B 0,C 180,E1 -1887.917,E2 -1887.917} C_VEL
LIN {X 0,Y 580.045,Z 481.936,A -85,B 0,C 180,E1 -1888.611,E2 -1888.611} C_VEL
LIN {X 0,Y 580.036,Z 482.711,A -85,B 0,C 180,E1 -1889.306,E2 -1889.306} C_VEL
LIN {X 0,Y 580.034,Z 483,A -85,B 0,C 180,E1 -1890,E2 -1890} C_VEL
LIN {X 0,Y 580.036,Z 482.711,A -85,B 0,C 180,E1 -1890.694,E2 -1890.694} C_VEL
LIN {X 0,Y 580.045,Z 481.936,A -85,B 0,C 180,E1 -1891.389,E2 -1891.389} C_VEL
LIN {X 0,Y 580.041,Z 480.681,A -85,B 0,C 180,E1 -1892.083,E2 -1892.083} C_VEL
LIN {X 0,Y 580.07,Z 477.788,A -85,B 0,C 180,E1 -1893.125,E2 -1893.125} C_VEL
LIN {X 0,Y 580.137,Z 475.148,A -85,B 0,C 180,E1 -1893.82,E2 -1893.82} C_VEL
LIN {X 0,Y 580.084,Z 469.986,A -85,B 0,C 180,E1 -1894.865,E2 -1894.865} C_VEL
LIN {X 0,Y 580.193,Z 463.188,A -85,B 0,C 180,E1 -1895.91,E2 -1895.91} C_VEL
LIN {X 0,Y 580.225,Z 455.497,A -85,B 0,C 180,E1 -1896.808,E2 -1896.808} C_VEL
LIN {X 0,Y 580.252,Z 448.409,A -85,B 0,C 180,E1 -1897.481,E2 -1897.481} C_VEL
LIN {X 0,Y 580.307,Z 440.549,A -85,B 0,C 180,E1 -1898.093,E2 -1898.093} C_VEL
LIN {X 0,Y 580.416,Z 430.735,A -85,B 0,C 180,E1 -1898.705,E2 -1898.705} C_VEL
LIN {X 0,Y 580.455,Z 419.307,A -85,B 0,C 180,E1 -1899.231,E2 -1899.231} C_VEL
LIN {X 0,Y 580.527,Z 409.254,A -85,B 0,C 180,E1 -1899.56,E2 -1899.56} C_VEL
LIN {X 0,Y 580.558,Z 400.456,A -85,B 0,C 180,E1 -1899.757,E2 -1899.757} C_VEL
LIN {X 0,Y 580.613,Z 332.557,A -85,B 0,C 180,E1 -1900.614,E2 -1900.614} C_VEL
LIN {X 0,Y 580.328,Z 324.995,A -85,B 0,C 180,E1 -1900.715,E2 -1900.715} C_VEL
LIN {X 0,Y 580.2,Z 323.456,A -85,B 0,C 180,E1 -1900.789,E2 -1900.789} C_VEL
LIN {X 0,Y 580.247,Z 309.514,A -85,B 0,C 180,E1 -1903.304,E2 -1903.304} C_VEL
LIN {X 0,Y 580.355,Z 295.85,A -85,B 0,C 180,E1 -1905.811,E2 -1905.811} C_VEL
LIN {X 0,Y 580.503,Z 280.234,A -85,B 0,C 180,E1 -1908.713,E2 -1908.713} C_VEL
LIN {X 0,Y 580.294,Z 273.138,A -85,B 0,C 180,E1 -1910.076,E2 -1910.076} C_VEL
LIN {X 0,Y 580.238,Z 273.009,A -85,B 0,C 180,E1 -1912.996,E2 -1912.996} C_VEL
LIN {X 0,Y 580.257,Z 273.018,A -85,B 0,C 180,E1 -1915.85,E2 -1915.85} C_VEL
LIN {X 0,Y 580.271,Z 273.013,A -85,B 0,C 180,E1 -1918.977,E2 -1918.977} C_VEL
LIN {X 0,Y 580.278,Z 273.012,A -85,B 0,C 180,E1 -1922.027,E2 -1922.027} C_VEL
LIN {X 0,Y 580.268,Z 273.012,A -85,B 0,C 180,E1 -1924.697,E2 -1924.697} C_VEL
LIN {X 0,Y 580.276,Z 273.02,A -85,B 0,C 180,E1 -1927.269,E2 -1927.269} C_VEL
LIN {X 0,Y 580.267,Z 273.011,A -85,B 0,C 180,E1 -1930.268,E2 -1930.268} C_VEL
LIN {X 0,Y 580.244,Z 273.017,A -85,B 0,C 180,E1 -1932.708,E2 -1932.708} C_VEL
LIN {X 0,Y 580.242,Z 273.017,A -85,B 0,C 180,E1 -1935.611,E2 -1935.611} C_VEL
LIN {X 0,Y 580.261,Z 273.016,A -85,B 0,C 180,E1 -1938.67,E2 -1938.67} C_VEL
LIN {X 0,Y 580.256,Z 273.023,A -85,B 0,C 180,E1 -1940.963,E2 -1940.963} C_VEL
LIN {X 0,Y 580.234,Z 273.016,A -85,B 0,C 180,E1 -1943.594,E2 -1943.594} C_VEL
LIN {X 0,Y 580.259,Z 273.013,A -85,B 0,C 180,E1 -1946.142,E2 -1946.142} C_VEL
LIN {X 0,Y 580.254,Z 273.02,A -85,B 0,C 180,E1 -1948.613,E2 -1948.613} C_VEL
LIN {X 0,Y 580.264,Z 273.017,A -85,B 0,C 180,E1 -1951.022,E2 -1951.022} C_VEL
LIN {X 0,Y 580.256,Z 273.013,A -85,B 0,C 180,E1 -1953.671,E2 -1953.671} C_VEL
LIN {X 0,Y 580.234,Z 273.023,A -85,B 0,C 180,E1 -1956.44,E2 -1956.44} C_VEL
LIN {X 0,Y 580.238,Z 273.015,A -85,B 0,C 180,E1 -1959.436,E2 -1959.436} C_VEL
LIN {X 0,Y 580.222,Z 273.017,A -85,B 0,C 180,E1 -1961.644,E2 -1961.644} C_VEL
LIN {X 0,Y 580.254,Z 273.02,A -85,B 0,C 180,E1 -1964.546,E2 -1964.546} C_VEL
LIN {X 0,Y 580.221,Z 273.021,A -85,B 0,C 180,E1 -1966.695,E2 -1966.695} C_VEL
LIN {X 0,Y 580.293,Z 273.01,A -85,B 0,C 180,E1 -1968.827,E2 -1968.827} C_VEL
LIN {X 0,Y 580.287,Z 273.011,A -85,B 0,C 180,E1 -1971.643,E2 -1971.643} C_VEL
LIN {X 0,Y 580.297,Z 273.013,A -85,B 0,C 180,E1 -1974.44,E2 -1974.44} C_VEL
LIN {X 0,Y 580.332,Z 273.011,A -85,B 0,C 180,E1 -1977.918,E2 -1977.918} C_VEL
LIN {X 0,Y 580.337,Z 273.012,A -85,B 0,C 180,E1 -1980,E2 -1980} C_VEL
LIN {X 0,Y 580.289,Z 273.009,A -85,B 0,C 180,E1 -1982.777,E2 -1982.777} C_VEL
LIN {X 0,Y 580.294,Z 273.013,A -85,B 0,C 180,E1 -1985.56,E2 -1985.56} C_VEL
LIN {X 0,Y 580.28,Z 273.012,A -85,B 0,C 180,E1 -1988.357,E2 -1988.357} C_VEL
LIN {X 0,Y 580.254,Z 273.015,A -85,B 0,C 180,E1 -1991.174,E2 -1991.174} C_VEL
LIN {X 0,Y 580.279,Z 273.014,A -85,B 0,C 180,E1 -1994.018,E2 -1994.018} C_VEL
LIN {X 0,Y 580.238,Z 273.016,A -85,B 0,C 180,E1 -1996.9,E2 -1996.9} C_VEL
LIN {X 0,Y 580.258,Z 273.018,A -85,B 0,C 180,E1 -1999.824,E2 -1999.824} C_VEL
LIN {X 0,Y 580.261,Z 273.018,A -85,B 0,C 180,E1 -2001.289,E2 -2001.289} C_VEL
LIN {X 0,Y 579.603,Z 273.107,A -85,B 0,C 180,E1 -2001.868,E2 -2001.868} C_VEL
LIN {X 0,Y 576.72,Z 273.464,A -85,B 0,C 180,E1 -2002.807,E2 -2002.807} C_VEL
LIN {X 0,Y 574.286,Z 273.764,A -85,B 0,C 180,E1 -2003.564,E2 -2003.564} C_VEL
LIN {X 0,Y 573.255,Z 273.886,A -85,B 0,C 180,E1 -2004.148,E2 -2004.148} C_VEL
LIN {X 0,Y 573.181,Z 273.894,A -85,B 0,C 180,E1 -2004.345,E2 -2004.345} C_VEL
LIN {X 0,Y 573.18,Z 273.898,A -85,B 0,C 180,E1 -2006.98,E2 -2006.98} C_VEL
LIN {X 0,Y 573.204,Z 273.891,A -85,B 0,C 180,E1 -2010.179,E2 -2010.179} C_VEL
LIN {X 0,Y 573.233,Z 273.889,A -85,B 0,C 180,E1 -2012.646,E2 -2012.646} C_VEL
LIN {X 0,Y 573.176,Z 273.904,A -85,B 0,C 180,E1 -2015.19,E2 -2015.19} C_VEL
LIN {X 0,Y 573.212,Z 273.891,A -85,B 0,C 180,E1 -2017.81,E2 -2017.81} C_VEL
LIN {X 0,Y 573.238,Z 273.889,A -85,B 0,C 180,E1 -2020.526,E2 -2020.526} C_VEL
LIN {X 0,Y 573.197,Z 273.893,A -85,B 0,C 180,E1 -2023.665,E2 -2023.665} C_VEL
LIN {X 0,Y 573.192,Z 273.898,A -85,B 0,C 180,E1 -2026.638,E2 -2026.638} C_VEL
LIN {X 0,Y 573.223,Z 273.89,A -85,B 0,C 180,E1 -2029.478,E2 -2029.478} C_VEL
LIN {X 0,Y 573.215,Z 273.892,A -85,B 0,C 180,E1 -2032.192,E2 -2032.192} C_VEL
LIN {X 0,Y 573.212,Z 273.892,A -85,B 0,C 180,E1 -2035.232,E2 -2035.232} C_VEL
LIN {X 0,Y 573.232,Z 273.888,A -85,B 0,C 180,E1 -2037.775,E2 -2037.775} C_VEL
LIN {X 0,Y 573.212,Z 273.899,A -85,B 0,C 180,E1 -2040.632,E2 -2040.632} C_VEL
LIN {X 0,Y 573.206,Z 273.891,A -85,B 0,C 180,E1 -2043.514,E2 -2043.514} C_VEL
LIN {X 0,Y 573.19,Z 273.899,A -85,B 0,C 180,E1 -2046.133,E2 -2046.133} C_VEL
LIN {X 0,Y 573.22,Z 273.894,A -85,B 0,C 180,E1 -2049.173,E2 -2049.173} C_VEL
LIN {X 0,Y 573.278,Z 274.002,A -85,B 0,C 180,E1 -2049.878,E2 -2049.878} C_VEL
LIN {X 0,Y 573.498,Z 279.998,A -85,B 0,C 180,E1 -2051.05,E2 -2051.05} C_VEL
LIN {X 0,Y 573.319,Z 295.61,A -85,B 0,C 180,E1 -2053.99,E2 -2053.99} C_VEL
LIN {X 0,Y 573.199,Z 311.222,A -85,B 0,C 180,E1 -2056.89,E2 -2056.89} C_VEL
LIN {X 0,Y 573.136,Z 323.561,A -85,B 0,C 180,E1 -2059.133,E2 -2059.133} C_VEL
LIN {X 0,Y 573.309,Z 325.32,A -85,B 0,C 180,E1 -2059.203,E2 -2059.203} C_VEL
LIN {X 0,Y 573.666,Z 329.3,A -85,B 0,C 180,E1 -2059.26,E2 -2059.26} C_VEL
LIN {X 0,Y 573.585,Z 400.423,A -85,B 0,C 180,E1 -2060.167,E2 -2060.167} C_VEL
LIN {X 0,Y 573.518,Z 410.897,A -85,B 0,C 180,E1 -2060.411,E2 -2060.411} C_VEL
LIN {X 0,Y 573.416,Z 422.583,A -85,B 0,C 180,E1 -2060.832,E2 -2060.832} C_VEL
LIN {X 0,Y 573.353,Z 432.973,A -85,B 0,C 180,E1 -2061.364,E2 -2061.364} C_VEL
LIN {X 0,Y 573.257,Z 441.152,A -85,B 0,C 180,E1 -2061.895,E2 -2061.895} C_VEL
LIN {X 0,Y 573.191,Z 448.909,A -85,B 0,C 180,E1 -2062.515,E2 -2062.515} C_VEL
LIN {X 0,Y 573.156,Z 457.134,A -85,B 0,C 180,E1 -2063.324,E2 -2063.324} C_VEL
LIN {X 0,Y 573.113,Z 464.132,A -85,B 0,C 180,E1 -2064.194,E2 -2064.194} C_VEL
LIN {X 0,Y 573.004,Z 469.742,A -85,B 0,C 180,E1 -2065.075,E2 -2065.075} C_VEL
LIN {X 0,Y 573.037,Z 474.955,A -85,B 0,C 180,E1 -2066.132,E2 -2066.132} C_VEL
LIN {X 0,Y 572.992,Z 477.641,A -85,B 0,C 180,E1 -2066.836,E2 -2066.836} C_VEL
LIN {X 0,Y 572.941,Z 480.579,A -85,B 0,C 180,E1 -2067.891,E2 -2067.891} C_VEL
LIN {X 0,Y 572.944,Z 481.873,A -85,B 0,C 180,E1 -2068.594,E2 -2068.594} C_VEL
LIN {X 0,Y 572.936,Z 482.689,A -85,B 0,C 180,E1 -2069.297,E2 -2069.297} C_VEL
LIN {X 0,Y 572.936,Z 482.996,A -85,B 0,C 180,E1 -2070,E2 -2070} C_VEL
LIN {X 0,Y 572.937,Z 482.73,A -85,B 0,C 180,E1 -2070.703,E2 -2070.703} C_VEL
LIN {X 0,Y 572.945,Z 481.996,A -85,B 0,C 180,E1 -2071.406,E2 -2071.406} C_VEL
LIN {X 0,Y 572.941,Z 480.784,A -85,B 0,C 180,E1 -2072.109,E2 -2072.109} C_VEL
LIN {X 0,Y 572.991,Z 477.936,A -85,B 0,C 180,E1 -2073.164,E2 -2073.164} C_VEL
LIN {X 0,Y 573.025,Z 475.342,A -85,B 0,C 180,E1 -2073.868,E2 -2073.868} C_VEL
LIN {X 0,Y 572.983,Z 470.233,A -85,B 0,C 180,E1 -2074.925,E2 -2074.925} C_VEL
LIN {X 0,Y 573.113,Z 464.735,A -85,B 0,C 180,E1 -2075.806,E2 -2075.806} C_VEL
LIN {X 0,Y 573.156,Z 456.34,A -85,B 0,C 180,E1 -2076.849,E2 -2076.849} C_VEL
LIN {X 0,Y 573.216,Z 448.921,A -85,B 0,C 180,E1 -2077.574,E2 -2077.574} C_VEL
LIN {X 0,Y 573.284,Z 441.167,A -85,B 0,C 180,E1 -2078.193,E2 -2078.193} C_VEL
LIN {X 0,Y 573.329,Z 432.993,A -85,B 0,C 180,E1 -2078.725,E2 -2078.725} C_VEL
LIN {X 0,Y 573.432,Z 422.604,A -85,B 0,C 180,E1 -2079.257,E2 -2079.257} C_VEL
LIN {X 0,Y 573.523,Z 410.931,A -85,B 0,C 180,E1 -2079.678,E2 -2079.678} C_VEL
LIN {X 0,Y 573.595,Z 400.481,A -85,B 0,C 180,E1 -2079.921,E2 -2079.921} C_VEL
LIN {X 0,Y 573.626,Z 343.228,A -85,B 0,C 180,E1 -2080.657,E2 -2080.657} C_VEL
LIN {X 0,Y 573.469,Z 326.451,A -85,B 0,C 180,E1 -2080.869,E2 -2080.869} C_VEL
LIN {X 0,Y 573.186,Z 323.852,A -85,B 0,C 180,E1 -2080.934,E2 -2080.934} C_VEL
LIN {X 0,Y 573.151,Z 321.471,A -85,B 0,C 180,E1 -2081.314,E2 -2081.314} C_VEL
LIN {X 0,Y 573.246,Z 305.852,A -85,B 0,C 180,E1 -2084.193,E2 -2084.193} C_VEL
LIN {X 0,Y 573.401,Z 290.233,A -85,B 0,C 180,E1 -2087.107,E2 -2087.107} C_VEL
LIN {X 0,Y 573.475,Z 276.568,A -85,B 0,C 180,E1 -2089.694,E2 -2089.694} C_VEL
LIN {X 0,Y 573.27,Z 273.991,A -85,B 0,C 180,E1 -2090.216,E2 -2090.216} C_VEL
LIN {X 0,Y 573.211,Z 273.885,A -85,B 0,C 180,E1 -2093.138,E2 -2093.138} C_VEL
LIN {X 0,Y 573.234,Z 273.889,A -85,B 0,C 180,E1 -2096.191,E2 -2096.191} C_VEL
LIN {X 0,Y 573.193,Z 273.892,A -85,B 0,C 180,E1 -2098.566,E2 -2098.566} C_VEL
LIN {X 0,Y 573.213,Z 273.892,A -85,B 0,C 180,E1 -2100.993,E2 -2100.993} C_VEL
LIN {X 0,Y 573.238,Z 273.896,A -85,B 0,C 180,E1 -2103.52,E2 -2103.52} C_VEL
LIN {X 0,Y 573.182,Z 273.895,A -85,B 0,C 180,E1 -2106.053,E2 -2106.053} C_VEL
LIN {X 0,Y 573.227,Z 273.89,A -85,B 0,C 180,E1 -2108.702,E2 -2108.702} C_VEL
LIN {X 0,Y 573.201,Z 273.896,A -85,B 0,C 180,E1 -2111.589,E2 -2111.589} C_VEL
LIN {X 0,Y 573.201,Z 273.894,A -85,B 0,C 180,E1 -2114.672,E2 -2114.672} C_VEL
LIN {X 0,Y 573.204,Z 273.894,A -85,B 0,C 180,E1 -2117.596,E2 -2117.596} C_VEL
LIN {X 0,Y 573.227,Z 273.891,A -85,B 0,C 180,E1 -2120.569,E2 -2120.569} C_VEL
LIN {X 0,Y 573.223,Z 273.897,A -85,B 0,C 180,E1 -2123.075,E2 -2123.075} C_VEL
LIN {X 0,Y 573.235,Z 273.888,A -85,B 0,C 180,E1 -2125.669,E2 -2125.669} C_VEL
LIN {X 0,Y 573.214,Z 273.891,A -85,B 0,C 180,E1 -2128.183,E2 -2128.183} C_VEL
LIN {X 0,Y 573.221,Z 273.897,A -85,B 0,C 180,E1 -2130.632,E2 -2130.632} C_VEL
LIN {X 0,Y 573.204,Z 273.891,A -85,B 0,C 180,E1 -2133.512,E2 -2133.512} C_VEL
LIN {X 0,Y 573.183,Z 273.896,A -85,B 0,C 180,E1 -2136.132,E2 -2136.132} C_VEL
LIN {X 0,Y 573.215,Z 273.891,A -85,B 0,C 180,E1 -2139.172,E2 -2139.172} C_VEL
LIN {X 0,Y 573.181,Z 273.894,A -85,B 0,C 180,E1 -2141.41,E2 -2141.41} C_VEL
LIN {X 0,Y 573.193,Z 273.902,A -85,B 0,C 180,E1 -2144.351,E2 -2144.351} C_VEL
LIN {X 0,Y 573.183,Z 273.901,A -85,B 0,C 180,E1 -2146.528,E2 -2146.528} C_VEL
LIN {X 0,Y 573.243,Z 273.886,A -85,B 0,C 180,E1 -2149.403,E2 -2149.403} C_VEL
LIN {X 0,Y 573.244,Z 273.896,A -85,B 0,C 180,E1 -2152.249,E2 -2152.249} C_VEL
LIN {X 0,Y 573.264,Z 273.884,A -85,B 0,C 180,E1 -2155.077,E2 -2155.077} C_VEL
LIN {X 0,Y 573.301,Z 273.886,A -85,B 0,C 180,E1 -2157.892,E2 -2157.892} C_VEL
LIN {X 0,Y 573.306,Z 273.888,A -85,B 0,C 180,E1 -2160,E2 -2160} C_VEL
LIN {X 0,Y 573.257,Z 273.885,A -85,B 0,C 180,E1 -2162.811,E2 -2162.811} C_VEL
LIN {X 0,Y 573.263,Z 273.889,A -85,B 0,C 180,E1 -2165.628,E2 -2165.628} C_VEL
LIN {X 0,Y 573.221,Z 273.89,A -85,B 0,C 180,E1 -2168.46,E2 -2168.46} C_VEL
LIN {X 0,Y 573.223,Z 273.892,A -85,B 0,C 180,E1 -2171.313,E2 -2171.313} C_VEL
LIN {X 0,Y 573.244,Z 273.887,A -85,B 0,C 180,E1 -2174.414,E2 -2174.414} C_VEL
LIN {X 0,Y 573.179,Z 273.897,A -85,B 0,C 180,E1 -2177.114,E2 -2177.114} C_VEL
LIN {X 0,Y 573.253,Z 273.891,A -85,B 0,C 180,E1 -2179.33,E2 -2179.33} C_VEL
LIN {X 0,Y 573.186,Z 273.894,A -85,B 0,C 180,E1 -2182.34,E2 -2182.34} C_VEL
LIN {X 0,Y 573.215,Z 273.899,A -85,B 0,C 180,E1 -2185.412,E2 -2185.412} C_VEL
LIN {X 0,Y 573.183,Z 273.894,A -85,B 0,C 180,E1 -2188.567,E2 -2188.567} C_VEL
LIN {X 0,Y 573.202,Z 273.897,A -85,B 0,C 180,E1 -2190.995,E2 -2190.995} C_VEL
LIN {X 0,Y 573.232,Z 273.892,A -85,B 0,C 180,E1 -2193.521,E2 -2193.521} C_VEL
LIN {X 0,Y 573.176,Z 273.895,A -85,B 0,C 180,E1 -2196.054,E2 -2196.054} C_VEL
LIN {X 0,Y 573.223,Z 273.893,A -85,B 0,C 180,E1 -2198.703,E2 -2198.703} C_VEL
LIN {X 0,Y 573.193,Z 273.895,A -85,B 0,C 180,E1 -2201.46,E2 -2201.46} C_VEL
LIN {X 0,Y 573.208,Z 273.892,A -85,B 0,C 180,E1 -2204.336,E2 -2204.336} C_VEL
LIN {X 0,Y 573.207,Z 273.893,A -85,B 0,C 180,E1 -2207.362,E2 -2207.362} C_VEL
LIN {X 0,Y 573.221,Z 273.893,A -85,B 0,C 180,E1 -2210.392,E2 -2210.392} C_VEL
LIN {X 0,Y 573.223,Z 273.893,A -85,B 0,C 180,E1 -2213.076,E2 -2213.076} C_VEL
LIN {X 0,Y 573.241,Z 273.887,A -85,B 0,C 180,E1 -2215.67,E2 -2215.67} C_VEL
LIN {X 0,Y 573.219,Z 273.893,A -85,B 0,C 180,E1 -2218.184,E2 -2218.184} C_VEL
LIN {X 0,Y 573.227,Z 273.896,A -85,B 0,C 180,E1 -2220.633,E2 -2220.633} C_VEL
LIN {X 0,Y 573.201,Z 273.891,A -85,B 0,C 180,E1 -2223.515,E2 -2223.515} C_VEL
LIN {X 0,Y 573.193,Z 273.899,A -85,B 0,C 180,E1 -2226.133,E2 -2226.133} C_VEL
